(* CoDeSys 2.3 project: cy-wg-05-005.pro *)
(* Title: cy-wg-05 - ClevergyAS *)
(* Author: Andrea Ravasio *)
(* Libraries: Standard.lib 2.12.10 14:48:34, Util.lib 18.5.10 15:14:28, Visual.lib 2.12.10 14:48:34, WagoLibIdent.lib 25.2.13 11:12:16, WagoLibStatus.lib 2.12.10 14:48:32, SysLibFile.lib 2.12.10 14:48:34, SysLibRtc.lib 2.12.10 14:48:32, SysLibSockets.lib 10.2.11 09:20:54, SysLibEvent.lib 2.12.10 14:48:34, SysLibPlcCtrl.lib 2.12.10 14:48:32, SysLibCallback.lib 2.12.10 14:48:32, mod_com.lib 2.12.10 14:48:32, SerComm.lib 31.5.11 08:54:36, Serial_Interface_01.lib 22.4.13 12:50:14, Modb_l05.lib 22.4.13 12:50:12, MBus_03.lib 9.2.13 17:51:58 *)

(* PLC configuration (modules and I/O channels)
K-Bus [K_Bus] node 0, in %IB0 out %QB0
  0750-0402 4 DI 24 V DC 3.0ms [Type_1_4_Channels] node 0, in %IB8 out %QB8 {INTTypePAAssignment = PLC; INTTypeModule = plugged}
    VPN_OUT2 AT %IX4.0 [BOOLOnX_I] Ch_1 Digital input
    KEY_QE_ST AT %IX4.1 [BOOLOnX_I] Ch_2 Digital input
    AT %IX4.2 [BOOLOnX_I] Ch_3 Digital input
    AT %IX4.3 [BOOLOnX_I] Ch_4 Digital input
  0750-0504 4 DO 24V DC 0.5A [Type_10_4_Channels] node 1, in %IB8 out %QB8 {INTTypePAAssignment = PLC; INTTypeModule = plugged}
    AT %QX4.0 [BOOLOnX_Q] Ch_1 Digital output
    AT %QX4.1 [BOOLOnX_Q] Ch_2 Digital output
    TEST1 AT %QX4.2 [BOOLOnX_Q] Ch_3 Digital output
    TEST2 AT %QX4.3 [BOOLOnX_Q] Ch_4 Digital output
  0750-0653/0003-0000#03 RS485 Interface (Adjustable), 3 Bytes [Type_21_1_Channels] node 2, in %IB4 out %QB4 {INTTypePAAssignment = PLC; INTTypeModule = plugged}
    AT %IX0.0 [BOOLOnX_I] Transmission acknowledgement
    AT %IX0.1 [BOOLOnX_I] Reception request
    AT %IX0.2 [BOOLOnX_I] Initialization acknowledgement
    AT %IX0.3 [BOOLOnX_I] Input buffer is full
    AT %IX0.4 [BOOLOnX_I] Number of received characters Bit 0
    AT %IX0.5 [BOOLOnX_I] Number of received characters Bit 1
    AT %IX0.6 [BOOLOnX_I] Number of received characters Bit 2
    AT %IB1 [BYTEOnB_I] Input data Byte 0
    AT %IB2 [BYTEOnB_I] Input data Byte 1
    AT %IB3 [BYTEOnB_I] Input data Byte 2
    AT %QX0.0 [BOOLOnX_Q] Transmission request
    AT %QX0.1 [BOOLOnX_Q] Reception acknowledgement
    AT %QX0.2 [BOOLOnX_Q] Initialization request
    AT %QX0.4 [BOOLOnX_Q] Number of characters Bit 0
    AT %QX0.5 [BOOLOnX_Q] Number of characters Bit 1
    AT %QX0.6 [BOOLOnX_Q] Number of characters Bit 2
    AT %QB1 [BYTEOnB_Q] Output data Byte 0
    AT %QB2 [BYTEOnB_Q] Output data Byte 1
    AT %QB3 [BYTEOnB_Q] Output data Byte 2
  0750-0650/0003-0000#03 RS 232 C Interface (Adjustable), 3 Byte [Type_21_1_Channels] node 0, in %IB4 out %QB4 {INTTypePAAssignment = PLC; INTTypeModule = plugged}
    AT %IX2.0 [BOOLOnX_I] Transmission acknowledgement
    AT %IX2.1 [BOOLOnX_I] Reception request
    AT %IX2.2 [BOOLOnX_I] Initialization acknowledgement
    AT %IX2.3 [BOOLOnX_I] Input buffer is full
    AT %IX2.4 [BOOLOnX_I] Number of received characters Bit 0
    AT %IX2.5 [BOOLOnX_I] Number of received characters Bit 1
    AT %IX2.6 [BOOLOnX_I] Number of received characters Bit 2
    AT %IB5 [BYTEOnB_I] Input data Byte 0
    AT %IB6 [BYTEOnB_I] Input data Byte 1
    AT %IB7 [BYTEOnB_I] Input data Byte 2
    AT %QX2.0 [BOOLOnX_Q] Transmission request
    AT %QX2.1 [BOOLOnX_Q] Reception acknowledgement
    AT %QX2.2 [BOOLOnX_Q] Initialization request
    AT %QX2.4 [BOOLOnX_Q] Number of characters Bit 0
    AT %QX2.5 [BOOLOnX_Q] Number of characters Bit 1
    AT %QX2.6 [BOOLOnX_Q] Number of characters Bit 2
    AT %QB5 [BYTEOnB_Q] Output data Byte 0
    AT %QB6 [BYTEOnB_Q] Output data Byte 1
    AT %QB7 [BYTEOnB_Q] Output data Byte 2
Fieldbus variables [FB_VARS] node 1, in %IB0 out %QB0
Flag variables [FLAG_VARS] node 2, in %IB0 out %QB0
Modbus-Master [MB_MASTER] node 3, in %IB0 out %QB0
*)

(* Global variable list: Global_Constants *)
VAR_GLOBAL CONSTANT

	Plant_NAME			: STRING :='cySN:5 cyVER:5 - Gavazzeni C Energetiche';
	Plant_SN			: DWORD  :=5;  		(* S/N Impianto di telecontrollo *)
	Plant_SW_VER		: WORD   :=5;		(* Versione SW installata *)

	(* Parameters *)
	Plant_DefaultTAmb	: INT	:=100;		(* [.1°C] Temperatura ambiente di default in caso di rottura sonda *)
	Plant_MaxRunTAmb	: INT   :=250; 		(* [.1°C] Temperatura ambiente massima funzionamento impianto *)
	Plant_AntiFreezeTAmb: INT   :=-40;		(* [.1°C] Antifreeze temperature, start circulators *)
	Plant_VRD_TAlarm	: INT   :=450; 		(* [.1°C] Temperatura di allarme VRD, blocco *)
	Plant_VRD_TMax		: INT   :=430; 		(* [.1°C] Setpoint massimo per uscita VRD *)
	Plant_VRD_TDefault	: INT	:=300;		(* [.1°C] Temperatura di default in caso di errore climatica *)
	Plant_CirOffDelay	: TIME	:=T#15m;	(* (Def.T#15m) Ritardo spegnimento pompe per ricircolo caldaia *)
	Plant_MaxWaterLoss	: WORD  :=2;		(* [lt/h] Massima perdita del circuito *)

	(* Filesystem *)
	FilesPath  			: STRING :='S:\';

	(* TCP Logger *)
	Logger_SERVER		: STRING:='';
	Logger_IP			: STRING:='192.168.100.3';
	Logger_PORT			: WORD  :=80;
	Logger_GETSTART		: STRING:='GET /cygmsrv/hsgm.ashx?';
	Logger_GETEND		: STRING:='$R$N$R$N';
	Logger_CHECK		: STRING:='True';
	Logger_CRLF			: STRING:='$R$N';
	Logger_DataFile		: STRING:='S:\LOG.DAT';
	Logger_DataFileOld	: STRING:='S:\LOG.BCK';
	Logger_IndexFile	: STRING:='S:\LOG.IDX';
	Logger_ConnRetries	: BYTE:=5;
	Logger_RecoverMsgs	: BYTE:=25;

	(* TCP Remote *)
	Remote_PORT			: WORD  :=10;
	Remote_WELCOME		: STRING:='Connected$R$N';
	Remote_OK			: STRING:='OK$R$N';
	Remote_ERROR		: STRING:='ERROR$R$N';

	(* TCP Sockets *)
	MAX_SEND_TCP_SERVER					 : DWORD:=1500;(*60000*)
	MAX_RECEIVE_TCP_SERVER				 : DWORD:=3000;
	MAX_RECEIVE_TCP_SERVER_SOCKET	 	 : DWORD:=1500;
	MAX_SEND_TCP_CLIENT					 : DWORD:=1500;(*15000*)
	MAX_RECEIVE_TCP_CLIENT				 : DWORD:=1500;
	MAX_RECEIVE_TCP_CLIENT_SOCKET		 : DWORD:=1500;
	MAX_RECEIVE_UDP_SERVER				 : INT  :=1472;
	MAX_RECEIVE_UDP_CLIENT				 : INT  :=1472;
	CONNECT_WATCHDOG_TIME				 : TIME :=t#10s;

END_VAR

(* Global variable list: Global_Retain *)
VAR_GLOBAL RETAIN PERSISTENT
	Mode_Manual : BOOL := FALSE;
END_VAR

(* Global variable list: Global_Variables *)
VAR_GLOBAL

	SYS    : typ_SYS;

	MODB01 : obj_MODBUS						:= ( ID:=1 , COM:=2, BAUDRATE:=BAUD_9600, RS485:=TRUE );
	GAS01  : obj_MODBUS_ELGAS_MINIELCOR		:= ( ID:=1 , ADDRESS:=1 );

	MBUS01 : obj_MBUS						:= ( ID:=1 , COM:=3, BAUDRATE:=BAUD_2400 );
	CTB01  : obj_MBUS_CTB_SHARKY775			:= ( ID:=1 , ADDRESS:=16#51311891 );
	CTB02  : obj_MBUS_CTB_SHARKY775			:= ( ID:=2 , ADDRESS:=16#51311893 );
	CTB03  : obj_MBUS_CTB_SHARKY775			:= ( ID:=3 , ADDRESS:=16#51311892 );
	CTB04  : obj_MBUS_CTB_SHARKY775			:= ( ID:=4 , ADDRESS:=16#51038660 );

	Logger : typ_Logger;

	(**** SIMULATION ONLY ****)
(*	VPN_ST2		:BOOL:=TRUE;
	KEY_QE_ST	:BOOL:=TRUE;
*)

END_VAR

(* Data type in Logger *)
TYPE en_Logger_ErrLev :
(
	EL_Log			:=0,
	EL_Wrn			:=1,
	EL_Alarm		:=2,
	EL_AlarmStop	:=3
);
END_TYPE

(* Data type in Logger *)
TYPE en_Logger_Status :
(
	S_Logger_UNKNOWN := 0,
	S_Logger_IDLE,
	S_Logger_WAITCONN,
	S_Logger_WAITTX,
	S_Logger_WAITRESP,
	S_Logger_ERROR
);
END_TYPE

(* Data type *)
TYPE en_SYS_Objects :
(
	EO_SYS		:=0,  (* PLC *)
	EO_VPN		:=1,  (* VPN *)
	EO_DOOR		:=2,  (* Door & access control *)

	EO_CAL		:=10, (* Caldaia *)
	EO_CIR		:=11, (* Circolatore *)
	EO_CRON		:=12, (* Crono-termostato *)
	EO_VRD		:=13, (* Valvola miscelatore pannelli *)
	EO_CTL		:=14, (* Contalitri *)
	EO_CTB		:=15, (* Contabilizzatore *)
	EO_TPV		:=16, (* Temperature probes values *)
	EO_PPV		:=17, (* Pressure probes values *)
	EO_PBV		:=18, (* Over-Pressure Alarms *)
	EO_TBV		:=19, (* Over-Temperature Alarms *)
	EO_PMV		:=20, (* Under-Pressure Alarms *)
	EO_GRU		:=21, (* Gruppo termico *)
	EO_PDC		:=22, (* Pompa di calore *)
	EO_SOL		:=23, (* Pannello solare termico *)
	EO_ESOL		:=24, (* Pannello solare fotovoltaico *)
	EO_GAS		:=25, (* Contatore GAS *)
	EO_PORT		:=26, (* Misuratore di portata *)
	EO_FPV		:=27, (* Flow probes value *)
	EO_ANZ		:=28, (* Analizzatore di rete elettrica *)

	EO_LON		:=1000, (* Bus - LON *)
	EO_MODBUS	:=1001, (* Bus - MODBUS *)
	EO_MBUS		:=1002  (* Bus - M-BUS *)
);
END_TYPE

(* Data type *)
TYPE en_SYS_Status :
(
	S_UNKNOWN  := 0,
	S_STARTUP,
	S_INIT_RTC,
	S_INIT_VAR,
	S_AUTOTEST,
	S_RUNNING,
	S_SHUTDOWN,
	S_HALT
);
END_TYPE

(* Data type in Plant_Objects *)
TYPE typ_Clima : (* CURVA CLIMATICA *)
STRUCT
	InitOK:		BOOL;
	Points: 	ARRAY [0..10] OF POINT;
END_STRUCT
END_TYPE

(* Data type in Plant_Objects *)
TYPE typ_Cron_Calendar :
STRUCT
	Profile		: ARRAY[0..384] OF BYTE;
END_STRUCT
END_TYPE

(* Data type in Plant_Objects *)
TYPE typ_Cron_Jolly :
STRUCT
	Start		: DT;
	End			: DT;
	Temp		: WORD;
	Flags		: WORD; (* B0:Enabled B1..B15:Unused *)
END_STRUCT
END_TYPE

(* Data type in Plant_Objects *)
TYPE typ_Cron_Profile :
STRUCT
	Flags		: WORD;
	Setpoint	: ARRAY [0..95] OF WORD;
END_STRUCT
END_TYPE

(* Data type in Logger *)
TYPE typ_Logger :
STRUCT
	Status		: en_Logger_Status;

	SendReq		: BOOL;
	SendIdx		: DWORD;
	SendData	: ARRAY [0..MAX_SEND_TCP_CLIENT] OF BYTE;
	SendLen		: DINT;

	TData		: ARRAY [0..MAX_SEND_TCP_CLIENT] OF BYTE;
	TLen		: DINT;

	LastIdxPos	: DWORD;

	(* Temporary variables used by objects *)
	s1			: STRING(256);
	i1			: WORD;

END_STRUCT
END_TYPE

(* Data type in Plant_Objects *)
TYPE typ_MODBUS_ABB_DMTME72 :
STRUCT
	V_3P		: DWORD; (* V *)
	V_L1N		: DWORD;
	V_L2N		: DWORD;
	V_L3N		: DWORD;
	V_L1L2		: DWORD;
	V_L2L3		: DWORD;
	V_L3L1		: DWORD;
	I_3P		: DWORD; (* 10^-3 A *)
	I_L1		: DWORD;
	I_L2		: DWORD;
	I_L3		: DWORD;
	PF_3P		: DINT;	 (* 10^-3 *)
	PF_L1		: DINT;
	PF_L2		: DINT;
	PF_L3		: DINT;
	COS_3P		: DINT;
	COS_L1		: DINT;
	COS_L2		: DINT;
	COS_L3		: DINT;
	VA_3P		: DWORD; (* VA *)
	VA_L1		: DWORD;
	VA_L2		: DWORD;
	VA_L3		: DWORD;
	P_3P		: DWORD; (* W *)
	P_L1		: DWORD;
	P_L2		: DWORD;
	P_L3		: DWORD;
	Q_3P		: DWORD; (* VAr *)
	Q_L1		: DWORD;
	Q_L2		: DWORD;
	Q_L3		: DWORD;

	WH_3P		: DWORD; (* 10^-2 Wh *)
	VARH_3P		: DWORD; (* 10^-2 VArh *)
	FREQ		: DWORD; (* 10^-3 Hz *)

	I_L1_Max	: DWORD;
	I_L2_Max	: DWORD;
	I_L3_Max	: DWORD;
	P_3P_Max	: DWORD;
	Q_3P_Max	: DWORD;
	P_3P_Avg15m	: DWORD;

END_STRUCT
END_TYPE

(* Data type in Plant_Objects *)
TYPE typ_MODBUS_ELGAS_MINIELCOR :
STRUCT
	Vb			: ARRAY [0..3] OF WORD;	(* m^3 *)
	Vm			: DWORD;				(* m^3 *)
	P			: REAL;					(* bar *)
	T			: REAL;					(* °C *)
	C			: REAL;
	Vbs			: ARRAY [0..3] OF WORD;	(* m^3 *)
	Vb_d_d		: ARRAY [0..3] OF WORD;	(* m^3 *)
	Vb_d_m		: ARRAY [0..3] OF WORD;	(* m^3 *)
	Vm_d_d		: DWORD;				(* m^3 *)
	Q			: REAL;					(* m^3/h *)
	Qb			: REAL;					(* m^3/h *)

	BC_EVC		: REAL;			(* % *)
	BV_EVC		: REAL;			(* V *)
	D_Err		: WORD;			(* 0:OK, 1:FAIL *)
	Status		: DWORD;		(* Status bits *)

END_STRUCT
END_TYPE

(* Data type in Plant_Objects *)
TYPE typ_MODBUS_FRER_IQ96U2 :
STRUCT
	V_L1N		: DWORD; (* 10^-3 V *)
	V_L2N		: DWORD;
	V_L3N		: DWORD;
	V_L1L2		: DWORD;
	V_L2L3		: DWORD;
	V_L3L1		: DWORD;
	I_L1		: DWORD; (* 10^-3 I *)
	I_L2		: DWORD;
	I_L3		: DWORD;
	FREQ		: DWORD; (* 10^-3 Hz *)
	P_3P		: DWORD; (* W *)
	Q_3P		: DWORD; (* VAr *)
	PF_3P		: DINT;	 (* 10^-3 *)
	WH_3P		: DWORD; (* Wh *)
	VARH_3P		: DWORD; (* VArh *)
	MULT		: DWORD;

	WH_3P_NEG	: DWORD; (* Wh *)
	VARH_3P_NEG : DWORD; (* VArh *)
	S_3P		: DWORD; (* VA *)

	PF_L1		: DWORD; (* 10^-3 *)
	PF_L2		: DWORD; (* 10^-3 *)
	PF_L3		: DWORD; (* 10^-3 *)

	P_3P_Max	: DWORD;
	P_3P_Avg15m	: DWORD;
	I_L1_Max	: DWORD;
	I_L2_Max	: DWORD;
	I_L3_Max	: DWORD;
	I_L1_Avg15m	: DWORD;
	I_L2_Avg15m	: DWORD;
	I_L3_Avg15m	: DWORD;

END_STRUCT
END_TYPE

(* Data type in Plant_Objects *)
TYPE typ_MODBUS_VAR : (* Gestione parametri MODBUS *)
STRUCT
	SlaveAddress	: BYTE;
	FunCode			: BYTE;
	FunAddress		: WORD;
	Refresh_Time	: BYTE; (* 0:No refresh x:Refresh in seconds *)
	Refresh_Cnt		: BYTE; (* INTERNAL *)
	Variable		: POINTER TO WORD;
	Variable_Size	: BYTE;
	Variable_Mirror : WORD; (* INTERNAL [Force refresh on read variables when <>0] *)
END_STRUCT
END_TYPE

(* Data type *)
TYPE typ_SYS :
STRUCT
	Status			: en_SYS_Status;
	Warning			: BOOL;
	Alarm			: BOOL;
	AlarmStop		: BOOL;

	Time_LogString	: STRING;
	Time_Year		: WORD;
	Time_Month		: BYTE;
	Time_Day		: BYTE;

	Time_CT_DT		: DT;
	Time_CT_Day		: WORD;
	Time_CT_Quarter	: BYTE;

	LastLogs_Idx	: BYTE;
	LastLogs_Dat	: ARRAY[0..5] OF STRING;
	LastLogs_Msg	: ARRAY[0..5] OF STRING;

END_STRUCT
END_TYPE

(* POU PLC_PRG, ST *)
PROGRAM PLC_PRG
VAR
	Timer1: TON; (* Fast controls tick *)
	Timer2: TON; (* Plant control tick *)
	Timer3: TON; (* Logger timer *)
END_VAR
(******************************************************************************
 ****                           MAIN TASK CODE                             ****
 ******************************************************************************

	Network setup:
		IP  = 192.168.100.2 | MSK = 255.255.255.0
		GW	= 192.168.100.1 | DNS = 192.168.100.1
		SNTP = 193.204.114.232 (3600s) ==> 192.168.100.3

*)

(*==============================*)
(*===== Main status machine ====*)
(*==============================*)
Main_Stm();

(*==============================*)
(*== Running cycle operations ==*)
(*==============================*)
IF SYS.Status>S_INIT_VAR THEN

	(* Execute MODBUS01 process *)
	MODB01();
	GAS01( MODBUS:=MODB01 );

	(* Execute MBUS01 process *)
	MBUS01();
	CTB01( MBUS:=MBUS01 );
	CTB02( MBUS:=MBUS01 );
	CTB03( MBUS:=MBUS01 );
	CTB04( MBUS:=MBUS01 );

END_IF

(*==============================*)
(*== System cycle operations ===*)
(*==============================*)
(* Execute TCP processes *)
Logger_Proc();
Remote_Proc();
(* Update user led *)
USRLED_Update();
(* Execute Cron Editor commands *)
(*CronEd(); *)
(* External resources *)
(*	IF NOT TPV01.ERR THEN T_AMB:=T_S01;
ELSIF NOT TPV05.ERR THEN T_AMB:=GRU01.TAmb;
ELSE 					 T_AMB:=Plant_DefaultTAmb;
END_IF *)

(**** SIMULATION ONLY ****)
(*...*)
END_PROGRAM
ACTION Main_Stm:
CASE Sys.Status OF

	S_STARTUP:
		Sys.Status:=S_INIT_RTC;

	S_INIT_RTC:
		(* Check RTC and update from network *)
		RTC_Update();
		(* Check time *)
		IF Sys.Time_Year>2000 THEN
			Sys.Status:=S_INIT_VAR;
		END_IF

	S_INIT_VAR:
		LogEv(EL_Wrn,EO_SYS,0,1,CONCAT('System_startup_v',WORD_TO_STRING(Plant_SW_VER)));
		Sys.Status:=S_RUNNING;

	S_RUNNING:
		Timer1(IN:=NOT Timer1.Q,PT:=T#50ms);
		IF Timer1.Q THEN
			(* Update meters *)

			(* Update system checks *)
			SYS_Proc();
		END_IF

		Timer2(IN:=NOT Timer2.Q,PT:=T#500ms);
		IF Timer2.Q THEN
			(* Read current date/time *)
			RTC_Update();
			(* Execute plant operations *)

			(* Test toggle *)
			IF TEST1 THEN TEST1:=FALSE; ELSE TEST1:=TRUE; END_IF
		END_IF

		Timer3(IN:=NOT Timer3.Q,PT:=T#5m);
		IF Timer3.Q THEN
			(* Trig logger *)
			LogTrig();
			(* Execute temporary CSV logger *)
			(*CSV_Log();*)
		END_IF

	S_SHUTDOWN:
		(* Stop sistema *)
		Sys.Status:=S_STARTUP;

	S_HALT:
		(* Aspetta uscita manuale *)
		Sys.Status:=S_STARTUP;

ELSE
	Sys.Status:=S_STARTUP;
END_CASE;
END_ACTION

(* POU TCP_Logger/Logger_Proc, ST *)
PROGRAM Logger_Proc
VAR
	c1:         	TCPCLIENT;

	Open:	    	BOOL;
	IpAddr:			DWORD;
	InetAddr:		DWORD;
	Connected:  	BOOL;
	Error:      	DINT;
	TxTrig:     	BOOL;
	RxData:			ARRAY [0..MAX_RECEIVE_TCP_CLIENT] OF BYTE;
	RxLen:			DINT;

	Retry:			BYTE;	(* Counter for connection retries *)
	Recovered:		BYTE;	(* Counter for recovered unsent messages *)

	i:				DINT;
	pos:			DWORD;
	hFile:			DWORD;

END_VAR
(*=== State machine ===*)
CASE Logger.Status OF

	S_Logger_UNKNOWN:
		(* Startup *)
		Logger.SendReq:=FALSE;
		Open:=FALSE;
		Logger.Status:=S_Logger_IDLE;

	S_Logger_IDLE:
		(* Wait request *)
		IF Logger.SendReq THEN
			(* Resolve server name or use static IP *)
			IF LEN(Logger_SERVER)=0 THEN
				InetAddr:=SysSockInetAddr(Logger_IP);
			ELSE
				IpAddr:=SysSockGetHostByName(ADR(Logger_SERVER));
				DWORDSWAP(pIn:=ADR(IpAddr), pOut:=ADR(InetAddr));
			END_IF
			TxTrig:=FALSE;
			RxLen:=0;
			(* Open connection *)
			Open:=TRUE;
			Logger.Status:=S_Logger_WAITCONN;
		END_IF

	S_Logger_WAITCONN:
		(* Wait connection *)
		IF Connected THEN
			(* Send data *)
			TxTrig:=TRUE;
			Logger.Status:=S_Logger_WAITTX;
		END_IF
		IF Error>0 THEN
			Open:=FALSE;
			Logger.Status:=S_Logger_ERROR;
		END_IF

	S_Logger_WAITTX:
		(* Wait transmission *)
		IF NOT TxTrig THEN
			Logger.Status:=S_Logger_WAITRESP;
		END_IF
		IF Error>0 THEN
			Open:=FALSE;
			Logger.Status:=S_Logger_ERROR;
		END_IF

	S_Logger_WAITRESP:
		(* Wait response *)
		IF Connected=FALSE (* OR TIMEOUT!! *) THEN
			Open:=FALSE;
			(* Check response *)
			IF RxLen>=4 AND CHKSTRING(pString:=ADR(RxData), pPattern:=ADR(Logger_CHECK)) THEN
				Logger.SendReq:=FALSE;
				Retry:=0;
				(* Check unsent messages to flush *)
				IF Recovered<Logger_RecoverMsgs THEN
					MsgChk();
					IF Logger.SendReq=TRUE THEN
						Recovered:=Recovered+1;
					ELSE
						Recovered:=0;
					END_IF
				ELSE
					Recovered:=0;
				END_IF
				Logger.Status:=S_Logger_IDLE;
			ELSE
				Logger.Status:=S_Logger_ERROR;
			END_IF
		END_IF

	S_Logger_ERROR:
		(* Connection error or send failure *)
		Retry:=Retry+1;
		IF Retry>Logger_ConnRetries THEN
			(* Save message as unsent *)
			MsgSave();
			Logger.SendReq:=FALSE;
			Retry:=0;
		END_IF
		Logger.Status:=S_Logger_IDLE;

ELSE
	Logger.Status:=S_Logger_UNKNOWN;
END_CASE


(*=== Execute client lib ===*)
c1(
	xOpenConnection			:= Open,
	dwInetAddr 				:= InetAddr,
	wPortNumber				:= Logger_PORT,
	ptSendData				:= ADR(Logger.SendData),
	diSendCount				:= Logger.SendLen,
	tConnectWatchdogTime	:= t#10s,
	xStartSend				:= TxTrig,
	aReceiveBuffer			:= RxData,
	diReceiveCount			:= RxLen,
	xConnected				=> Connected,
	diError					=> Error
);

(*=== Process Rx data ===*)
(*IF RxLen>0 THEN
	RxLen:=0;
END_IF*)
END_PROGRAM
ACTION MsgChk:
(* Open index file *)
hFile:=SysFileOpen(Logger_IndexFile,'r');
IF hFile=0 THEN
	RETURN;
END_IF
(* Search oldest message to recover *)
SysFileSetPos(hFile,Logger.LastIdxPos);
Logger.SendLen:=0;
REPEAT
	SysFileRead(hFile, ADR(Logger.SendIdx), SIZEOF(Logger.SendIdx));
	pos:=SysFileGetPos(hFile);
	SysFileRead(hFile, ADR(Logger.SendLen), SIZEOF(Logger.SendLen));
UNTIL
	SysFileEOF(hFile) OR Logger.SendLen<>0
END_REPEAT
SysFileClose(hFile);
(* Delete index file when all messages are recovered *)
IF Logger.SendLen=0 THEN
	Logger.LastIdxPos:=0;
	SysFileDelete(Logger_IndexFile);
	RETURN;
END_IF
(* Recover message data *)
hFile:=SysFileOpen(Logger_DataFile,'r');
IF hFile<>0 THEN
	SysFileSetPos(hFile,Logger.SendIdx);
	SysFileRead(hFile,ADR(Logger.SendData),Logger.SendLen);
	Logger.SendReq:=TRUE;
	SysFileClose(hFile);
END_IF
(* Clear index entry *)
hFile:=SysFileOpen(Logger_IndexFile,'a');
IF hFile<>0 THEN
	SysFileSetPos(hFile,pos);
	i:=0;
	SysFileWrite(hFile, ADR(i), 4);
	Logger.LastIdxPos:=SysFileGetPos(hFile);
	SysFileClose(hFile);
END_IF
END_ACTION
ACTION MsgSave:
(* Add log position in recovery indexes *)
hFile:=SysFileOpen(Logger_IndexFile,'a');
SysFileWrite(hFile, ADR(Logger.SendIdx), SIZEOF(Logger.SendIdx));
SysFileWrite(hFile, ADR(Logger.SendLen), SIZEOF(Logger.SendLen));
SysFileClose(hFile);
END_ACTION

(* POU Utils Functions/TCPCLIENT, ST *)
FUNCTION_BLOCK TCPCLIENT
(***********************************************************************************************************	*)
(* Version: 1.3b                        			          													*)
(* Date: 28.10.2014                   				          							            			*)
(***********************************************************************************************************	*)
(* WAGO Kontakttechnik GmbH Hansastr. 27 32423 Minden(Westf.)													*)
(* Tel. +0049 571/887-0 Fax. +0049 571/887-0																	*)
(* Author: VB																									*)
(***********************************************************************************************************	*)
(*Description:	A TCP client to read and write data with additional connection watchdog							*)
(*History:																										*)
(*Version 1.3b: 28.10.2014: Use DWORD address for IP (Andrea Ravasio)											*)
(*Version 1.3: 11.02.2011: Changes according to 750-880/881											 			*)
(*Version 1.2: 29.08.2007 Bugfix TCP Client																		*)
(*Version 1.1: 15.01.2007 Changes according to FW11																*)
(*Version 1.0: 09.03.2006 Release																				*)
(***********************************************************************************************************	*)
VAR CONSTANT
	STATE_CREATE     				 : BYTE:= 0;
	STATE_OPEN     					 : BYTE:= 1;
	STATE_IOCTL    					 : BYTE:= 2;
	STATE_CONNECT     				 : BYTE:= 10;
	STATE_TX       					 : BYTE:= 20;
	STATE_RX       					 : BYTE:= 30;
	STATE_CLOSE    					 : BYTE:= 40;
	STATE_ERROR_TRAP			     : BYTE:= 200;
END_VAR

VAR_INPUT
	xOpenConnection					: BOOL;
	dwInetAddr						: DWORD; (* <== Use SysSockInetAddr() value or
													swapped bytes order of SysSockGetHostByName() value *)
	wPortNumber						: WORD;
	ptSendData						: POINTER TO ARRAY[0..MAX_SEND_TCP_CLIENT] OF BYTE;
	diSendCount						: DINT;
	tConnectWatchdogTime		    : TIME := t#10s;
END_VAR
VAR_OUTPUT
	xConnected						: BOOL;
	diError 						: DINT := 0;
END_VAR
(* ErrorCodes -----------------------------------------
	16#8001 => No socket descriptor available 
	16#8002 => SysSockSend returns -1 
	16#8003 => Socket was "gracefully closed" 
	16#8004 => switching to none blocking mode fails
	16#8005 => SysSockClose() returns FALSE 
    16#8006 => SysSockConnect() fails
    16#8007 => SysSockSend() fails
	16#8008 => error state machine 
	16#8009 => timeout while waiting for data from server 
------------------------------------------------------------*)
VAR_IN_OUT
	xStartSend							: BOOL;
	aReceiveBuffer						: ARRAY [0..MAX_RECEIVE_TCP_CLIENT] OF BYTE;
	diReceiveCount						: DINT;
END_VAR
VAR
	m_State								: BYTE := 0;
	m_ReceiveBuffer						: ARRAY [0..MAX_RECEIVE_TCP_CLIENT_SOCKET] OF BYTE;
	m_Socket							: DINT;
	m_AddressInfo						: SOCKADDRESS;
	m_BytesReceived						: DINT;
	m_diReturn							: DINT;
	m_xReturn							: BOOL;
	m_IoCtlParameter  					: DINT := 1; (* IOCTL-Parameter for non-blocking mode of sockets *)
	i									: INT;
	T_Connect							: TON;
	m_count								: DINT;
	diOption							: DINT := 1;
	m_Blocking   						: DINT := 0;
END_VAR
IF xOpenConnection THEN
	(* State maschine *)
	CASE  m_State OF

	(* -------------------------------------------------------------------------*)
	STATE_CREATE:
			(* create socket descriptor*)
			m_Socket := SysSockCreate(diAddressFamily	:= SOCKET_AF_INET,
													 diType		:= SOCKET_STREAM,
													 diProtocol := SOCKET_IPPROTO_TCP);
			IF m_Socket >= 0 THEN
			(*Set Push-Bit*)
				IF ADR(%MW0)=16#30000000  OR ADR(%MW0)=16#20000000 THEN (*841 or 881*)
					SysSockSetOption(
						diSocket:=m_Socket,
						diLevel:=6,
						diOption:=SOCKET_TCP_NODELAY,
						pOptionValue:=ADR(diOption),
						diOptionLength:=SIZEOF(diOption));
				ELSE
						;
				END_IF
				m_State := STATE_IOCTL; (* succesful *)
			ELSE
				diError := 16#8001;  (* no socket descriptor available *)
				m_State := STATE_ERROR_TRAP;
			END_IF

	(* -------------------------------------------------------------------------*)
	STATE_IOCTL: (* change  socket mode  to none blocking *)
		m_diReturn := SysSockIoctl( m_Socket, SOCKET_FIONBIO, ADR(m_IoCtlParameter));
		IF m_diReturn <> 0 THEN
			m_AddressInfo.sin_family := SOCKET_AF_INET;
			m_AddressInfo.sin_port := SysSockNtohs(wPortNumber);
			m_AddressInfo.sin_addr := dwInetAddr;
			m_State := STATE_CONNECT;
		ELSE
			diError := 16#8004;  (* switching to none blocking mode fails *)
			m_State := STATE_ERROR_TRAP;
		END_IF


	(* -------------------------------------------------------------------------*)
	STATE_CONNECT: (* connect with server *)
		T_Connect(IN:=TRUE , PT:=tConnectWatchdogTime);(*activate watchdog for establishing connection to a server*)
		m_xReturn := SysSockConnect ( m_Socket, ADR(m_AddressInfo),  SIZEOF(m_AddressInfo));
		IF m_xReturn THEN (* succesful *)
			IF xStartSend THEN
				m_State := STATE_TX;(*transmit data*)
			ELSE
				m_State := STATE_RX;(*wait for data from server*)
			END_IF
			xConnected:=TRUE;
			T_Connect(IN:=FALSE);
		ELSE
			IF T_Connect.Q THEN
				diError := 16#8006;  (* connect fails *)
				xConnected:=FALSE;
				T_Connect(IN:=FALSE);
				m_State := STATE_ERROR_TRAP;
				SysSockClose( m_Socket);
			ELSE
				m_State := STATE_CONNECT;(*client still  tries to set up connection*)
			END_IF
		END_IF


	STATE_TX:	 (* send TCP-message *)
		m_diReturn := SysSockSend(diSocket := m_Socket,
								  pbyBuffer := ADR(ptSendData^[0]),
								  diBufferSize := diSendCount-m_count,
								  diFlags := 0);

		CASE m_diReturn OF
		-1:	(* ERROR *)
			T_Connect(IN:=TRUE , PT:=CONNECT_WATCHDOG_TIME);(*activate watchdog to check communication*)
			IF t_Connect.Q THEN
				diError := 16#8007;
				T_Connect(IN:=FALSE);
				m_State:=STATE_CLOSE;
			END_IF
		0: (* socket was "gracefully closed" *)
			m_State := STATE_CLOSE;
			diError := 16#8003;
		ELSE (* succesful *)
			m_count:=m_count+m_diReturn;
			IF m_count>=diSendCount THEN
				diError := 16#0000;
				m_State := STATE_RX;
				m_count:=0;
				xStartSend:=FALSE;
			END_IF
			T_Connect(IN:=FALSE);
		END_CASE

	(* -------------------------------------------------------------------------*)
	STATE_RX: (* process receive data *)
			m_BytesReceived := SysSockRecv(	diSocket 	:= m_Socket,
										pbyBuffer 	:= ADR(m_ReceiveBuffer),		(* Address of receive buffer *)
										diBufferSize:= SIZEOF(m_ReceiveBuffer),
										diFlags		:= 0);

			CASE m_BytesReceived OF
			-1:	(* No data available or error occured *)
				T_Connect(IN:=TRUE , PT:=tConnectWatchdogTime);(*activate watchdog to check communication*)
				IF t_Connect.Q THEN
					diError:=16#8009;
					T_Connect(IN:=FALSE);
					m_State:=STATE_CLOSE;
				END_IF
				IF xStartSend THEN
					m_State:=STATE_TX	;(* WAIT IN THIS STATE  and check for arriving data or new send command*)
				END_IF;
			0: (* socket was "gracefully closed"  *)
				m_State:=STATE_CLOSE;
				diError := 16#8003;
			ELSE (* succesful *)
				diError := 16#0000;
				T_Connect(IN:=FALSE);
				(* Copy received data into receive buffer *)
				FOR i:= 0 TO DINT_TO_INT(m_BytesReceived	)-1 DO
					aReceiveBuffer[diReceiveCount]:= m_ReceiveBuffer[i];
					diReceiveCount:=(diReceiveCount+1) MOD SIZEOF(aReceiveBuffer);
				END_FOR

			END_CASE

	(* -------------------------------------------------------------------------*)
	STATE_CLOSE : (* close socket *)
		IF ADR(%MW0)=16#30000000  OR ADR(%MW0)=16#20000000 THEN (*841 or 881*)
			;
		ELSE
			SysSockShutdown(m_Socket, 0);;(*870*)
		END_IF
		m_xReturn := SysSockClose( m_Socket);
		m_Socket := -1;
		m_State := 0; (* succesful *)
		xConnected:=FALSE;
		T_Connect(IN:=FALSE);
	(* -------------------------------------------------------------------------*)
	STATE_ERROR_TRAP: (* error handling *)
		xConnected:=FALSE;

	ELSE  (* Bad FSM code trap  *)
			m_State:= STATE_ERROR_TRAP;
			diError:= 16#8008;
	END_CASE

ELSE(*close connection*)
	IF m_Socket >= 0 THEN
		IF ADR(%MW0)=16#30000000  OR ADR(%MW0)=16#20000000 THEN (*841 or 881*)
			;
		ELSE
			SysSockShutdown(m_Socket, 0);;(*870*)
		END_IF
		SysSockClose( m_Socket);
	END_IF
	m_Socket := -1;
	diError := 16#0000;
	m_State := STATE_CREATE;
	xConnected:=FALSE;
	T_Connect(IN:=FALSE);
END_IF
END_FUNCTION_BLOCK

(* POU Utils Functions/DWORDSWAP, ST *)
FUNCTION DWORDSWAP:BOOL
VAR_INPUT
	pIn:POINTER TO ARRAY[1..4] OF BYTE;
	pOut:POINTER TO ARRAY[1..4] OF BYTE;
END_VAR
VAR
END_VAR
pOut^[1]:=pIn^[4];
pOut^[2]:=pIn^[3];
pOut^[3]:=pIn^[2];
pOut^[4]:=pIn^[1];
END_FUNCTION

(* POU Utils Functions/CHKSTRING, ST *)
FUNCTION CHKSTRING : BOOL
VAR_INPUT
	pString: POINTER TO BYTE;
	pPattern: POINTER TO BYTE;
END_VAR
VAR
END_VAR
CHKSTRING:=TRUE;
WHILE pPattern^<>0 AND CHKSTRING DO
	IF pPattern^<>pString^ THEN CHKSTRING:=FALSE; END_IF
	pString:=pString+1;
	pPattern:=pPattern+1;
END_WHILE
END_FUNCTION

(* POU TCP_Remote/Remote_Proc, ST *)
PROGRAM Remote_Proc
VAR
	s1:         	TCPSERVER;
	Enable: 		BOOL;
	Connected: 		BOOL;
	Error: 			DINT;

	TxData:			ARRAY [0..MAX_SEND_TCP_SERVER] OF BYTE;
	TxLen:			DINT;
	TxTrig:			BOOL;

	RxData:			ARRAY [0..MAX_RECEIVE_TCP_SERVER] OF BYTE;
	RxLen:			DINT;

	Status:			DINT;

	(* Command interpreter *)

	Cmd_Buf:		ARRAY [0..MAX_RECEIVE_TCP_SERVER] OF BYTE;
	Cmd_Buf_U16:	POINTER TO WORD;
	Cmd_Buf_INT:	POINTER TO INT;
	Cmd_BufLen:		WORD;
	Cmd_St:			WORD;

	Cmd_Obj:		WORD;
	Cmd_ObjIdx:		WORD;
	Cmd_C:			WORD;
	Cmd_R:			WORD;
	Cmd_CLen:		WORD;
	Cmd_RLen:		WORD;

	i : WORD;
	j : INT;

END_VAR
(*=== State machine ===*)
CASE Status OF
	0: (* Startup *)
		TxLen:=0; TxTrig:=FALSE;
		RxLen:=0;
		Enable:=TRUE;
		Status:=1;

	1: (* Wait incoming connection *)
		IF Connected THEN
			(* Log access *)
			LogEv(EL_Log,EO_VPN,1,5,'Remote');
			(* Send welcome message *)
			ADDSTRING(pTxData:=ADR(TxData), pString:=ADR(Remote_WELCOME), TxLen:=TxLen);
			TxTrig:=TRUE;
			Cmd_BufLen:=0;
			Cmd_St:=0;
			Status:=2;
		END_IF
		IF Error>1 THEN
			Enable:=FALSE;
			Status:=0;
		END_IF

	2: (* Wait command *)
		IF RxLen>0 THEN
			(*=== Interpreter start ===*)
			IF Cmd_BufLen+(RxLen/2)>=MAX_RECEIVE_TCP_SERVER THEN
				(* ERROR *)
				Cmd_BufLen:=0;
			ELSE
				i:=HEXTORAW(pString:=ADR(RxData), StringLen:=DINT_TO_WORD(RxLen), pData:=ADR(Cmd_Buf[Cmd_BufLen]));
				Cmd_BufLen:=Cmd_BufLen+i;
			END_IF
			IF Cmd_BufLen>=8 THEN
				Cmd_Buf_U16:=ADR(Cmd_Buf[6]);
				IF Cmd_BufLen>=(8+Cmd_Buf_U16^) THEN
					Cmd_CLen:=Cmd_Buf_U16^;
					Cmd_Buf_U16:=ADR(Cmd_Buf[0]); Cmd_Obj:=Cmd_Buf_U16^;
					Cmd_Buf_U16:=ADR(Cmd_Buf[2]); Cmd_ObjIdx:=Cmd_Buf_U16^;
					Cmd_Buf_U16:=ADR(Cmd_Buf[4]); Cmd_C:=Cmd_Buf_U16^;
					Command();
					Cmd_BufLen:=0;
				END_IF
			END_IF
			(*=== Interpreter end ===*)
			RxLen:=0;
		END_IF
		IF NOT Connected THEN
			Status:=0;
		END_IF

ELSE
	Status:=0;
END_CASE


(*=== Execute server lib ===*)
s1(
	xEnable				:= Enable,
	wPortNumber			:= Remote_PORT,
	tServerTimeOut		:= t#15m,
	ptSendData			:= ADR(TxData),
	diSendCount			:= TxLen,
	xStartSend			:= TxTrig,
	aReceiveBuffer		:= RxData,
	diReceiveCount		:= RxLen,
	xClientConnected	=> Connected,
	diError				=> Error
);
END_PROGRAM
ACTION Cmd_CAL:
(* Check index *)(*
IF Cmd_ObjIdx<1 OR Cmd_ObjIdx>2 THEN
	Cmd_R:=2;
	RETURN;
END_IF

(* Process command *)
CASE Cmd_C OF

	3: (* TRY REARM *)
		IF Cmd_ObjIdx=1 THEN
			CAL01.Rearm:=TRUE;
		ELSE
			CAL02.Rearm:=TRUE;
		END_IF

ELSE
	Cmd_R:=3;
END_CASE
*);
END_ACTION
ACTION Cmd_CRON:
(* Check index *)(*
IF Cmd_ObjIdx<1 OR Cmd_Obj=2 OR Cmd_ObjIdx>6 THEN
	Cmd_R:=2;
	RETURN;
END_IF

(* Process command *)
CASE Cmd_C OF

	1: (* GET PROFILE *)
		IF Cmd_CLen<>3 THEN
			Cmd_R:=4;
		ELSE
			(* Load profile *)
			CronEd.CN_Sel:=WORD_TO_BYTE(Cmd_ObjIdx);
			Cmd_Buf_U16:=ADR(Cmd_Buf[8]);
			CronEd.CN_YSel:=Cmd_Buf_U16^;
			CronEd.PR_Sel:=Cmd_Buf[10];
			CronEd.PR_Load_Exe();
			(* Copy data *)
			Cmd_RLen:=192;
			TxLen:=TxLen+RAWTOHEX(ADR(CronEd.PR.Setpoint),192,ADR(TxData[TxLen]));
		END_IF

	2: (* SET PROFILE *)
		IF Cmd_CLen<>(3+192) THEN
			Cmd_R:=4;
		ELSE
			(* Save profile *)
			CronEd.CN_Sel:=WORD_TO_BYTE(Cmd_ObjIdx);
			Cmd_Buf_U16:=ADR(Cmd_Buf[8]);
			CronEd.CN_YSel:=Cmd_Buf_U16^;
			CronEd.PR_Sel:=Cmd_Buf[10];
			MEMCPY(ADR(Cmd_Buf[11]),ADR(CronEd.PR.Setpoint),192);
			CronEd.PR_Save_Exe();
		END_IF

	5: (* GET CALENDAR MONTH *)
		IF Cmd_CLen<>3 THEN
			Cmd_R:=4;
		ELSE
			(* Load calendar *)
			CronEd.CN_Sel:=WORD_TO_BYTE(Cmd_ObjIdx);
			Cmd_Buf_U16:=ADR(Cmd_Buf[8]);
			CronEd.CN_YSel:=Cmd_Buf_U16^;
			CronEd.CA_Sel:=Cmd_Buf[10];
			CronEd.CA_Load_Exe();
			(* Copy data *)
			Cmd_RLen:=32;
			TxLen:=TxLen+RAWTOHEX(ADR(CronEd.CA.Profile),32,ADR(TxData[TxLen]));
		END_IF

	6: (* SET CALENDAR MONTH *)
		IF Cmd_CLen<>(3+32) THEN
			Cmd_R:=4;
		ELSE
			(* Save calendar *)
			CronEd.CN_Sel:=WORD_TO_BYTE(Cmd_ObjIdx);
			Cmd_Buf_U16:=ADR(Cmd_Buf[8]);
			CronEd.CN_YSel:=Cmd_Buf_U16^;
			CronEd.CA_Sel:=Cmd_Buf[10];
			MEMCPY(ADR(Cmd_Buf[11]),ADR(CronEd.CA.Profile),32);
			CronEd.CA_Save_Exe();
		END_IF

ELSE
	Cmd_R:=3;
END_CASE
*);
END_ACTION
ACTION Cmd_GRU:
(* Check index *)(*
IF Cmd_ObjIdx<>1 THEN
	Cmd_R:=2;
	RETURN;
END_IF

(* Process command *)
CASE Cmd_C OF

	1: (* GET CLIMATIC *)
		Cmd_RLen:=20;
		FOR i:=0 TO 4 DO
			j:=DINT_TO_INT(GRU01_Clima.Points[i].X);
			TxLen:=TxLen+RAWTOHEX(ADR(j),2,ADR(TxData[TxLen]));
			j:=DINT_TO_INT(GRU01_Clima.Points[i].Y);
			TxLen:=TxLen+RAWTOHEX(ADR(j),2,ADR(TxData[TxLen]));
		END_FOR

	2: (* SET CLIMATIC *)
		IF Cmd_CLen<>20 THEN
			Cmd_R:=4;
		ELSE
			FOR i:=0 TO 4 DO
				Cmd_Buf_INT:=ADR(Cmd_Buf[8+4*i]); j:=Cmd_Buf_INT^;
				GRU01_Clima.Points[i].X:=INT_TO_DINT(j);
				Cmd_Buf_INT:=ADR(Cmd_Buf[10+4*i]); j:=Cmd_Buf_INT^;
				GRU01_Clima.Points[i].Y:=INT_TO_DINT(j);
			END_FOR
		END_IF

ELSE
	Cmd_R:=3;
END_CASE
*);
END_ACTION
ACTION Cmd_PDC:
;(* Check index *)(*
IF Cmd_ObjIdx<>1 THEN
	Cmd_R:=2;
	RETURN;
END_IF

(* Process command *)
CASE Cmd_C OF

	3: (* TRY REARM *)
		PDC01.Rearm:=TRUE;

ELSE
	Cmd_R:=3;
END_CASE
*);
END_ACTION
ACTION Cmd_SYS:
(* Check index *)
IF Cmd_ObjIdx<>0 THEN
	Cmd_R:=2;
	RETURN;
END_IF

(* Process command *)
CASE Cmd_C OF

	0: (* ECHO *)
		IF Cmd_CLen<>0 THEN
			TxLen:=0;
		END_IF

	1: (* LOG REQUEST *)
		LogTrig();

	2: (* REARM *)
		Sys.Warning:=FALSE;
		Sys.Alarm:=FALSE;
		Sys.AlarmStop:=FALSE;

	3: (* GET INFO1 *)
		Cmd_RLen:=6;
		TxLen:=TxLen+RAWTOHEX(ADR(Plant_SN),4,ADR(TxData[TxLen]));
		TxLen:=TxLen+RAWTOHEX(ADR(Plant_SW_VER),2,ADR(TxData[TxLen]));

ELSE
	Cmd_R:=3;
END_CASE
END_ACTION
ACTION Command:
(* Default response OK/NODATA *)
Cmd_R:=0;
Cmd_RLen:=0;
TxLen:=16;

(* Check object *)
CASE Cmd_Obj OF

	EO_SYS:
		Cmd_SYS();
(*
	EO_GRU:
		Cmd_GRU();

	EO_PDC:
		Cmd_PDC();

	EO_CAL:
		Cmd_CAL();

	EO_CRON:
		Cmd_CRON();
*)
ELSE
	Cmd_R:=1;
END_CASE

(* Generate response *)
IF TxLen>0 THEN
	RAWTOHEX(ADR(Cmd_Obj)	,2,ADR(TxData[ 0]));
	RAWTOHEX(ADR(Cmd_ObjIdx),2,ADR(TxData[ 4]));
	RAWTOHEX(ADR(Cmd_R)		,2,ADR(TxData[ 8]));
	RAWTOHEX(ADR(Cmd_RLen)	,2,ADR(TxData[12]));
	TxTrig:=TRUE;
END_IF
END_ACTION

(* POU Utils Functions/TCPSERVER, ST *)
FUNCTION_BLOCK TCPSERVER
(***********************************************************************************************************	*)
(* Version: 1.6                                    			          											*)
(* Date: 11.02.2011                                   					          							    *)
(***********************************************************************************************************	*)
(* WAGO Kontakttechnik GmbH Hansastr. 27 32423 Minden(Westf.)													*)
(* Tel. +0049 571/887-0 Fax. +0049 571/887-0																	*)
(* Author: VB																									*)
(***********************************************************************************************************	*)
(*Description:	A TCP server to read and write data													       		*)
(*Historie:																										*)
(*Version 1.6: 11.02.2011: Changes according to 750-880/881											 			*)
(*Version 1.5: 27.11.2008 Bugfix allow reuse port																*)
(*Version 1.4: 13.10.2008 Bugfix transmitting large data														*)
(*Version 1.3: 15.01.2007 Changes according to FW11																*)
(*Version 1.2: 09.03.2006 Changes for socket handle 0											       			*)
(*Version 1.1: 14.02.2005 Release																				*)
(***********************************************************************************************************	*)
VAR CONSTANT
	STATE_INIT     				 : BYTE:= 0;
	STATE_OPEN     				 : BYTE:= 1;
	STATE_TX       				 : BYTE:= 20;
	STATE_RX       				 : BYTE:= 30;
	STATE_CLOSE    				 : BYTE:= 40;
	STATE_ERROR_TRAP		 	 : BYTE:= 200;
END_VAR
VAR_INPUT
	xEnable    					: BOOL;	 (* Set TRUE to enable function block *)
	wPortNumber					: WORD;  (* Port *)
	tServerTimeOut				: TIME:=t#50s;
	ptSendData					: POINTER TO ARRAY[0..MAX_SEND_TCP_SERVER] OF BYTE;
	diSendCount					: DINT;
END_VAR
VAR_OUTPUT
	xClientConnected  			: BOOL:= FALSE;
	diError 					: DINT:= 0;
END_VAR
(* Status Codes -----------------------------------------
	16#8001 => No socket descriptor available 
	16#8002 => SysSockBind fails 
	16#8003 => SysSockListen fails 
	16#8004 => switching to none blocking mode fails
	16#8005 => SysSockClose() returns FALSE 
    16#8006 => SysSockConnect() fails
    16#8007 => SysSockSend() fails
	16#8008 => error state machine 
	16#8009 => timeout while waiting for data from server 
	16#0001 => server waiting for client to establish connection
------------------------------------------------------------*)
VAR_IN_OUT
	xStartSend					: BOOL;
	aReceiveBuffer				: ARRAY [0..MAX_RECEIVE_TCP_SERVER] OF BYTE;
	diReceiveCount				: DINT;
END_VAR

VAR
	m_State    					: BYTE:= 0;
	m_ReceiveBuffer				: ARRAY [0..MAX_RECEIVE_TCP_SERVER_SOCKET] OF BYTE;
	m_ServerSocket				: DINT:= SOCKET_INVALID;
	m_Socket					: DINT:= SOCKET_INVALID;
	m_AddressInfo				: SOCKADDRESS;
	m_BytesReceived				: DINT;
	m_diReturn					: DINT;
	m_xReturn					: BOOL;
	m_SizeSockadr				: DWORD;
	m_ConnectionWatchdog		: TON;
	m_Flags						: DINT;
	m_NoneBlocking   			: DINT:= 1;
	m_Blocking   				: DINT:= 0;
	i							: INT;
	m_count						: DINT;
	diOption					: DINT := 1;
	on: DINT;
END_VAR
IF xEnable THEN
	CASE m_State OF
		STATE_INIT:
			(* Create Socket *)
			m_ServerSocket:= SysSockCreate( SOCKET_AF_INET, SOCKET_STREAM, 0);
			IF m_ServerSocket = SOCKET_INVALID THEN
				(* *)
				diError:= 16#8001;
				m_State:= STATE_ERROR_TRAP;
				RETURN;
			ELSE
				;
			END_IF
			(* Address bindings *)
			(********************)
			on:=1;
			SysSockSetOption( m_ServerSocket, SOCKET_SOL, SOCKET_SO_REUSEADDR, ADR(on), SIZEOF(on) );

			m_AddressInfo.sin_family:= SOCKET_AF_INET;
			m_AddressInfo.sin_port  := SysSockHtons( wPortNumber);
			m_AddressInfo.sin_addr  := SOCKET_INADDR_ANY;
			IF NOT SysSockBind( m_ServerSocket, ADR(m_AddressInfo), SIZEOF(m_AddressInfo)) THEN
				diError:= 16#8002;
				m_State:= STATE_ERROR_TRAP;
				RETURN;
			END_IF
			(* Wait for connections *)
			(************************)
			IF NOT SysSockListen( m_ServerSocket, 1) THEN
				diError:= 16#8003;
				m_State:= STATE_ERROR_TRAP;
			END_IF

			(* Puts SOCKET in NonBlocking mode *)
			m_diReturn:= SysSockIoctl( m_ServerSocket, SOCKET_FIONBIO, ADR(m_NoneBlocking));

			m_State:= STATE_OPEN;


		STATE_OPEN: 	(* Waiting for incomming connection *)
				m_SizeSockadr:=SIZEOF(m_AddressInfo);
				m_Socket:= SysSockAccept( m_ServerSocket, ADR(m_AddressInfo), ADR(m_SizeSockadr));
				diError:=State_open;
				IF m_Socket <> SOCKET_INVALID THEN
					xClientConnected:=TRUE;
					(*Set Push-Bit:new V1.5*)
					IF ADR(%MW0)=16#30000000  OR ADR(%MW0)=16#20000000 THEN (*841 or 881*)
						SysSockSetOption(
							diSocket:=m_Socket,
							diLevel:=6,
							diOption:=SOCKET_TCP_NODELAY,
							pOptionValue:=ADR(diOption),
							diOptionLength:=SIZEOF(diOption));
					ELSE
							;
					END_IF
					SysSockIoctl( m_Socket, SOCKET_FIONBIO, ADR(m_NoneBlocking));
					m_State:= STATE_RX;
					diError:=0;
				END_IF

		STATE_RX:
					m_BytesReceived:= SysSockRecv( m_Socket, ADR(m_ReceiveBuffer), SIZEOF(m_ReceiveBuffer), 0);
					CASE m_BytesReceived OF
					-1:(*no data available or error occured*)
						m_ConnectionWatchdog(IN:=TRUE , PT:=tServerTimeOut );
						IF m_connectionWatchdog.Q THEN
							m_State:= STATE_CLOSE;
							m_ConnectionWatchdog(IN:=FALSE);(*reset connection watchdog*)
							diError := 16#8009;
						END_IF
					0:(* socket was "gracefully closed"  *)
						m_State:= STATE_CLOSE;
						diError := 16#8003;
					ELSE
						(* Copy received data into receive buffer *)
						(********************************)
						FOR i:= 0 TO DINT_TO_INT(m_BytesReceived	)-1 DO
							aReceiveBuffer[diReceiveCount]:= m_ReceiveBuffer[i];
							diReceiveCount:=(diReceiveCount+1) MOD SIZEOF(aReceiveBuffer);
						END_FOR

						m_ConnectionWatchdog(IN:=FALSE);(*reset connection watchdog*)
					END_CASE

				(*send data*)
				IF xStartSend	 THEN
					m_State := STATE_TX;
				END_IF

	STATE_TX:	 (* send TCP-message *)
		m_diReturn := SysSockSend(diSocket := m_Socket,
								  pbyBuffer := ADR(ptSendData^[m_count]),(*geändert V1.4 bisher: [0] *)
								  diBufferSize := diSendCount-m_count,
								  diFlags :=m_Flags);
		CASE m_diReturn OF
		-1:	(* ERROR or data could not yet be send (V1.3 due to new FW11) *)
			m_ConnectionWatchdog(IN:=TRUE , PT:=tServerTimeOut );
			IF m_connectionWatchdog.Q THEN
				m_State:= STATE_CLOSE;
				m_ConnectionWatchdog(IN:=FALSE);(*reset connection watchdog*)
				diError := 16#8007;
			END_IF
		0: (* socket was "gracefully closed"  *)
			m_State := STATE_CLOSE;
			diError := 16#8003;
		ELSE (* succesful *)
			m_count:=m_count+m_diReturn;
			IF m_count>=diSendCount THEN
				diError := 16#0000;
				m_State := STATE_RX;
				m_count:=0;
				xStartSend:=FALSE;
			END_IF
			m_ConnectionWatchdog(IN:=FALSE);(*reset connection watchdog*)
		END_CASE


		STATE_CLOSE:	(* Close the server *)

		IF ADR(%MW0)=16#30000000  OR ADR(%MW0)=16#20000000 THEN (*841 or 881*)
			;
		ELSE
			IF m_Socket>=0 THEN
				SysSockShutdown(m_Socket, 0);;(*870*)
			END_IF
		END_IF
		IF m_Socket>=0 THEN
			SysSockClose( m_Socket);
		END_IF
		xClientConnected:= FALSE;
		m_State:= STATE_OPEN; (* Try to open the server again *)
		m_ConnectionWatchdog(IN:=FALSE);(*reset connection watchdog*)

		STATE_ERROR_TRAP: (* Error Read/Write socket  *)
			m_State:= STATE_ERROR_TRAP;

	ELSE  (* Bad FSM code trap  *)
			m_State:= STATE_ERROR_TRAP;
			diError:= 16#8008;
	END_CASE;
ELSE
	IF m_State <> STATE_INIT THEN
		IF ADR(%MW0)=16#30000000  OR ADR(%MW0)=16#20000000 THEN (*841 or 881*)
			;
		ELSE
			IF m_Socket>=0 THEN
				SysSockShutdown(m_Socket, 0);;(*870*)
			END_IF
		END_IF
		IF m_Socket>=0 THEN
			SysSockClose( m_Socket);
		END_IF
		IF ADR(%MW0)=16#30000000  OR ADR(%MW0)=16#20000000 THEN (*841 or 881*)
			;
		ELSE
			IF m_ServerSocket>=0 THEN
				SysSockShutdown(m_ServerSocket, 0);;(*870*)
			END_IF
		END_IF
		IF m_ServerSocket>=0 THEN
			SysSockClose( m_ServerSocket);
		END_IF
		xClientConnected:= FALSE;
		diError:= 0;
		m_State:= STATE_init; (* Try to open the server again *)
		m_ConnectionWatchdog(IN:=FALSE);(*reset connection watchdog*)
	END_IF
END_IF
END_FUNCTION_BLOCK

(* POU TCP_Logger/LogEv, ST *)
FUNCTION LogEv : BOOL
VAR_INPUT
	Level	: en_Logger_ErrLev;
	Object  : en_SYS_Objects;
	Index	: WORD;
	Error	: WORD;
	Message : STRING;
END_VAR
VAR
	s1 : STRING(160);
	i  : INT;
END_VAR
(* Execute error level operations *)
CASE Level OF
	EL_Wrn: 		Sys.Warning:=TRUE;
	EL_Alarm: 		Sys.Alarm:=TRUE;
	EL_AlarmStop: 	Sys.Alarm:=TRUE; (* GO TO STOP STATE!! *)
END_CASE

(* Fill lastlog list *)
s1:=CONCAT(Sys.Time_LogString,';Lev=');
s1:=CONCAT(s1,INT_TO_STRING(Level));
s1:=CONCAT(s1,';Obj=');
s1:=CONCAT(s1,INT_TO_STRING(Object));
s1:=CONCAT(s1,';Idx=');
s1:=CONCAT(s1,WORD_TO_STRING(Index));
s1:=CONCAT(s1,';Err=');
s1:=CONCAT(s1,WORD_TO_STRING(Error));
Sys.LastLogs_Dat[Sys.LastLogs_Idx]:=s1;
Sys.LastLogs_Msg[Sys.LastLogs_Idx]:=Message;
Sys.LastLogs_Idx:=Sys.LastLogs_Idx+1;
IF Sys.LastLogs_Idx>5 THEN Sys.LastLogs_Idx:=0; END_IF

(*---------------------------------------------------------------*)
(*---------------------------------------------------------------*)
Logger.TLen:=0;
(* Set GET header *)
ADDSTRING(ADR(Logger.TData), ADR(Logger_GETSTART), Logger.TLen);

(* Insert Header *)
s1:=INSERT('ID=&V=1&D=',DWORD_TO_STRING(Plant_SN),3);
s1:=CONCAT(s1,Sys.Time_LogString);
s1:=CONCAT(s1,'&S=');
IF Sys.Alarm THEN i:=2; ELSIF Sys.Warning THEN i:=1; ELSE i:=0; END_IF
s1:=CONCAT(s1,INT_TO_STRING(i));
ADDSTRING(ADR(Logger.TData), ADR(s1), Logger.TLen);

(* Insert ERR *)
s1:=CONCAT('&ERR=',INT_TO_STRING(Level));
s1:=CONCAT(s1,';');
s1:=CONCAT(s1,INT_TO_STRING(Object));
s1:=CONCAT(s1,';');
s1:=CONCAT(s1,WORD_TO_STRING(Index));
s1:=CONCAT(s1,';');
s1:=CONCAT(s1,WORD_TO_STRING(Error));
s1:=CONCAT(s1,';');
ADDSTRING(ADR(Logger.TData), ADR(s1), Logger.TLen);
s1:=Message;
STR_NOSPACES(ADR(s1));
ADDSTRING(ADR(Logger.TData), ADR(s1), Logger.TLen);

(* Finalize string *)
ADDSTRING(ADR(Logger.TData), ADR(Logger_GETEND), Logger.TLen);

(*---------------------------------------------------------------*)
(*---------------------------------------------------------------*)

Logger_Send();
END_FUNCTION

(* POU Utils Functions/ADDSTRING, ST *)
FUNCTION ADDSTRING : BOOL (* Append string to a byte buffer *)
VAR_INPUT
	pTxData: POINTER TO BYTE;
	pString: POINTER TO BYTE;
END_VAR
VAR_IN_OUT
	TxLen: DINT;
END_VAR
VAR
END_VAR
pTxData:=pTxData+TxLen;
WHILE pString^<>0 DO
	pTxData^:=pString^;
	pString:=pString+1;
	pTxData:=pTxData+1;
	TxLen:=TxLen+1;
END_WHILE
END_FUNCTION

(* POU Utils Functions/STR_NOSPACES, ST *)
FUNCTION STR_NOSPACES : BOOL (* Replace spaces and bad chars with allowed ones, used as HTTP-GET validator *)
VAR_INPUT
	pString: POINTER TO BYTE;
END_VAR
VAR
END_VAR
WHILE pString^<>0 DO
	IF pString^=16#20 (* space *) THEN pString^:=16#5F; (*'_'*) END_IF
	pString:=pString+1;
END_WHILE
END_FUNCTION

(* POU TCP_Logger/Logger_Send, ST *)
FUNCTION Logger_Send : BOOL
VAR
	hFile: 	DWORD;
	pos:	DWORD;
END_VAR
(* Read log position *)
pos:=SysFileGetSize(Logger_DataFile);
(* Check log size, bckup and erase if no pending messages *)
IF pos>100000000 (*100M*) THEN
	hFile:=SysFileOpen(Logger_IndexFile,'r');
	IF hFile=0 THEN
		SysFileDelete(Logger_DataFileOld);
		SysFileRename(Logger_DataFile,Logger_DataFileOld);
		pos:=0;
	ELSE
		SysFileClose(hFile);
	END_IF
END_IF
(* Write message on log file *)
hFile:=SysFileOpen(Logger_DataFile,'a');
IF hFile<>0 THEN
	SysFileWrite(hFile, ADR(Logger.TData), Logger.TLen);
	SysFileClose(hFile);
ELSE
	Sys.Warning:=TRUE;
END_IF


(* Check logger status *)
IF Logger.SendReq=FALSE THEN
	(* Set log position for recovery *)
	Logger.SendIdx:=pos;
	(* Copy message data *)
	MEMCPY(ADR(Logger.TData),ADR(Logger.SendData),DINT_TO_WORD(Logger.TLen));
	Logger.SendLen:=Logger.TLen;
	(* Trigger request *)
	Logger.SendReq:=TRUE;
ELSE
	(* Add message position+size in recovery indexes *)
	hFile:=SysFileOpen(Logger_IndexFile,'a');
	SysFileWrite(hFile, ADR(pos), SIZEOF(pos));
	SysFileWrite(hFile, ADR(Logger.TLen), SIZEOF(Logger.TLen));
	SysFileClose(hFile);
END_IF
END_FUNCTION

(* POU Utils Functions/MEMCPY, ST *)
FUNCTION MEMCPY:BOOL
VAR_INPUT
	pSourceAddress:POINTER TO ARRAY[1..2] OF BYTE;
	pDestinationAddress:POINTER TO ARRAY[1..2] OF BYTE;
	BytesToCopy:WORD;
END_VAR
VAR
END_VAR
WHILE (BytesToCopy > 0) DO
	pDestinationAddress^[1]:=pSourceAddress^[1]; (* copy bytes from source to destination *)
	pDestinationAddress:=ADR(pDestinationAddress^[2]); (* increment destination *)
	pSourceAddress:=ADR(pSourceAddress^[2]);(* increment source *)
	BytesToCopy:=BytesToCopy -1; (* decrement number of bytes to copy *)
END_WHILE
END_FUNCTION

(* POU Utils Functions/HEXTORAW, ST *)
FUNCTION HEXTORAW : WORD
VAR_INPUT
	pString		: POINTER TO BYTE;
	StringLen	: WORD;
	pData		: POINTER TO BYTE;
END_VAR
VAR
	xl: WORD;
	xi: WORD;
	xr: BYTE;
END_VAR
xl:=0;
xi:=0;

WHILE xi<StringLen DO

	IF pString^>=97 AND pString^<=102 THEN
		xr := pString^ - 87;
	ELSIF pString^>=65 AND pString^<=70 THEN
		xr := pString^ - 55;
	ELSIF pString^>=48 AND pString^<=57 THEN
		xr := pString^ - 48;
	ELSE
		xr := 16;
	END_IF

	IF xr<16 THEN
		IF (xi AND 1)=0 THEN
			pData^ := xr * 16;
		ELSE
			pData^ := pData^ + xr;
			pData := pData + 1;
			xl := xl + 1;
		END_IF
	END_IF

	xi := xi + 1;
	pString := pString + 1;

END_WHILE

HEXTORAW:=xl;
END_FUNCTION

(* POU Utils Functions/RAWTOHEX, ST *)
FUNCTION RAWTOHEX : WORD
VAR_INPUT
	pData: POINTER TO BYTE;
	DataLen: WORD;
	pString: POINTER TO BYTE;
END_VAR
VAR
	xl: WORD;
END_VAR
xl:=0;

WHILE DataLen>0 DO

	pString^ := (pData^ / 16#10) + 48 + (((pData^ / 16#10)/10)*7);
	pString:=pString+1;
	pString^ := (pData^ AND 16#0F)  + 48 + (((pData^ AND 16#0F)/10)*7);
	pString:=pString+1;
	pData:=pData+1;
	DataLen:=DataLen-1;
	xl:=xl+2;

END_WHILE

(*pString^:=0;*)

RAWTOHEX:=xl;
END_FUNCTION

(* POU Utils/USRLED_Update, ST *)
PROGRAM USRLED_Update
VAR
	OldStatus: en_SYS_Status;

	aFS : ARRAY [0..24] OF FLASHING_SEQUENCE :=
		(Colour:=GREEN,  Frequency:=1,   Relation:=128, Duration:=t#0s,    NextIndex:=0),  (* 0 => RUNNING *)
		(Colour:=ORANGE, Frequency:=1,   Relation:=128, Duration:=t#0s,    NextIndex:=1),  (* 1 => INIT *)
		(Colour:=RED,    Frequency:=4,   Relation:=128, Duration:=t#0s,    NextIndex:=2),  (* 2 => ERROR *)
		(Colour:=RED,    Frequency:=10,  Relation:=128, Duration:=t#0s,    NextIndex:=3),  (* 3 => ALARM *)
		(Colour:=ORANGE, Frequency:=200, Relation:=16,  Duration:=t#100ms, NextIndex:=11), (* 10 *)
		(Colour:=ORANGE, Frequency:=200, Relation:=32,  Duration:=t#100ms, NextIndex:=12),
		(Colour:=ORANGE, Frequency:=200, Relation:=64,  Duration:=t#100ms, NextIndex:=13),
		(Colour:=ORANGE, Frequency:=200, Relation:=128, Duration:=t#100ms, NextIndex:=14),
		(Colour:=ORANGE, Frequency:=200, Relation:=192, Duration:=t#100ms, NextIndex:=15),
		(Colour:=ORANGE, Frequency:=200, Relation:=128, Duration:=t#100ms, NextIndex:=16),
		(Colour:=ORANGE, Frequency:=200, Relation:=64,  Duration:=t#100ms, NextIndex:=17),
		(Colour:=ORANGE, Frequency:=200, Relation:=32,  Duration:=t#100ms, NextIndex:=18),
		(Colour:=ORANGE, Frequency:=200, Relation:=16,  Duration:=t#100ms, NextIndex:=19),
		(Colour:=ORANGE, Frequency:=200, Relation:=8,   Duration:=t#100ms, NextIndex:=10),
		(Colour:=GREEN,  Frequency:=200, Relation:=16,  Duration:=t#100ms, NextIndex:=21), (* 20 *)
		(Colour:=GREEN,  Frequency:=200, Relation:=32,  Duration:=t#100ms, NextIndex:=22),
		(Colour:=GREEN,  Frequency:=200, Relation:=64,  Duration:=t#100ms, NextIndex:=23),
		(Colour:=GREEN,  Frequency:=200, Relation:=128, Duration:=t#100ms, NextIndex:=24),
		(Colour:=GREEN,  Frequency:=200, Relation:=192, Duration:=t#100ms, NextIndex:=25),
		(Colour:=GREEN,  Frequency:=200, Relation:=128, Duration:=t#100ms, NextIndex:=26),
		(Colour:=GREEN,  Frequency:=200, Relation:=64,  Duration:=t#100ms, NextIndex:=27),
		(Colour:=GREEN,  Frequency:=200, Relation:=32,  Duration:=t#100ms, NextIndex:=28),
		(Colour:=GREEN,  Frequency:=200, Relation:=16,  Duration:=t#100ms, NextIndex:=29),
		(Colour:=GREEN,  Frequency:=200, Relation:=8,   Duration:=t#100ms, NextIndex:=20);

	pFS : POINTER TO FLASHING_SEQUENCE;


END_VAR
IF Sys.Status <> OldStatus THEN

	OldStatus:=Sys.Status;

	CASE OldStatus OF

		S_STARTUP:
			pFS:=ADR(aFS);
			SET_FLASHING_SEQUENCE(EN:=TRUE, POINTER_TO_POINTER_TO_ARRAY:=ADR(pFS));
			SET_FLASHING_SEQUENCE_INDEX(EN:=TRUE, IMMEDIATE:=FALSE, INDEX:=1);
			START_FLASHING_SEQUENCE(EN:=TRUE);

		S_RUNNING:
			SET_FLASHING_SEQUENCE_INDEX(EN:=TRUE, IMMEDIATE:=TRUE, INDEX:=0);

	END_CASE

END_IF
END_PROGRAM

(* POU Utils/CSV_Log, ST *)
FUNCTION CSV_Log : BOOL
VAR_INPUT
END_VAR
VAR CONSTANT
	LogFileName:STRING:='S:\LOGS_ID4V3.CSV';
END_VAR
VAR
	s1 : STRING(256);
	hFile: 	DWORD;
END_VAR
(* Check file presence *)
hFile:=SysFileOpen(LogFileName,'r');
IF hFile=0 THEN
	(*** File not exist *** Create file and write header *)
	hFile:=SysFileOpen(LogFileName,'w');
	IF hFile<>0 THEN
		(* Write CSV header *)
		s1:='DATE-TIME;T-Amb;T-GRU01-SetP;T-GRU01-Send;T-GRU01-Ret;T-GRU01-Amb;T_S01;T_S02;F-PDC01-Flow;T-PDC01-Send;T-PDC01-Ret;';
		SysFileWrite(hFile, ADR(s1), LEN(s1));
		s1:='T-CTB01-Send;T-CTB01-Ret;F-CTB01-Flow;P-CTB01-Power;E-CTB01-Energy';
		SysFileWrite(hFile, ADR(s1), LEN(s1));
		SysFileWrite(hFile, ADR(Logger_CRLF), LEN(Logger_CRLF));
	END_IF
ELSE
	(*** File exist *** Close file and reopen in append mode *)
	SysFileClose(hFile);
	hFile:=SysFileOpen(LogFileName,'a');
END_IF

(* Log to file *)
IF hFile<>0 THEN
	(* Date stamp *)
	s1:=REPLACE( Sys.Time_LogString , ' ' , 1 , 11 );
	SysFileWrite(hFile, ADR(s1), LEN(s1));
	(* Log data 1 *)
	s1:=CONCAT(';', INT_TO_STRING(T_AMB) );
	s1:=CONCAT(s1 , ';');
	s1:=CONCAT(s1 , INT_TO_STRING(GRU01.ActSetPoint) );
	s1:=CONCAT(s1 , ';');
	s1:=CONCAT(s1 , INT_TO_STRING(GRU01.TSend) );
	s1:=CONCAT(s1 , ';');
	s1:=CONCAT(s1 , INT_TO_STRING(GRU01.TRet) );
	s1:=CONCAT(s1 , ';');
	s1:=CONCAT(s1 , INT_TO_STRING(GRU01.TAmb) );
	s1:=CONCAT(s1 , ';');
	s1:=CONCAT(s1 , INT_TO_STRING(T_S01) );
	s1:=CONCAT(s1 , ';' );
	s1:=CONCAT(s1 , INT_TO_STRING(T_S02) );
	s1:=CONCAT(s1 , ';' );
	s1:=CONCAT(s1 , WORD_TO_STRING(PDC01.Flow) );
	s1:=CONCAT(s1 , ';' );
	s1:=CONCAT(s1 , INT_TO_STRING(PDC01.TSend) );
	s1:=CONCAT(s1 , ';');
	s1:=CONCAT(s1 , INT_TO_STRING(PDC01.TRet) );
	SysFileWrite(hFile, ADR(s1), LEN(s1));
	(* Log data 2 *)
	s1:=CONCAT(';', CTB01.M1.utFTemp.Value );
	s1:=CONCAT(s1 , ';');
	s1:=CONCAT(s1 , CTB01.M1.utRTemp.Value );
	s1:=CONCAT(s1 , ';');
	s1:=CONCAT(s1 , CTB01.M1.utFlow.Value );
	s1:=CONCAT(s1 , ';');
	s1:=CONCAT(s1 , CTB01.M1.utPower.Value );
	s1:=CONCAT(s1 , ';');
	s1:=CONCAT(s1 , CTB01.M1.utEnergy.Value );
	SysFileWrite(hFile, ADR(s1), LEN(s1));
	(* Add line CRLF and close *)
	SysFileWrite(hFile, ADR(Logger_CRLF), LEN(Logger_CRLF));
	SysFileClose(hFile);
END_IF
END_FUNCTION

(* POU Plant/SYS_Proc, ST *)
PROGRAM SYS_Proc
VAR
(*	fALARM_PB		:FLT_TAP;
	fALARM_TB		:FLT_TAP;
	fALARM_PM		:FLT_TAP; *)

(*	fGZB_ST			:FLT_TAP; (* GATEWAY ZIGBEE *)*)
(*	fVPN_OUT1		:FLT_TAP; (* VPN - CONNECT *)*)
	fVPN_OUT2		:FLT_TAP; (* VPN - STATUS *)
(*	fKEY_CT_ST		:FLT_TAP; (* DOOR01 - Porta primaria *)*)
(*	fKEY_SCT_ST		:FLT_TAP; (* DOOR02 - Porta secondaria *)*)
	fKEY_QE_ST		:FLT_TAP; (* DOOR03 - Quadro Elettrico *)

END_VAR
(*************** ISPESL *****************)
(*
fALARM_PB(IN:=ALARM_PB);
IF fALARM_PB.EVH THEN
	LogEv(EL_AlarmStop,EO_PBV,1,1,'Over_Pressure_Alarm');
END_IF

fALARM_TB(IN:=ALARM_TB);
IF fALARM_TB.EVH THEN
	LogEv(EL_AlarmStop,EO_TBV,1,1,'Over_Temperature_Alarm');
END_IF

fALARM_PM(IN:=ALARM_PM);
IF fALARM_PM.EVH THEN
	LogEv(EL_AlarmStop,EO_PMV,1,1,'Under_Pressure_Alarm');
END_IF
*)
(****************************************)

(*### VPN Connection Check ###*)(*
fVPN_OUT1(IN:=VPN_OUT1);
IF fVPN_OUT1.EVH THEN
	LogEv(EL_Log,EO_VPN,1,1,'CONNECT_ON');
END_IF
IF fVPN_OUT1.EVL THEN
	LogEv(EL_Log,EO_VPN,1,2,'CONNECT_OFF');
END_IF*)

(*### VPN Status Check ###*)
fVPN_OUT2(IN:=VPN_OUT2);
IF fVPN_OUT2.EVH THEN
	LogEv(EL_Log,EO_VPN,1,3,'STATUS_UP');
END_IF
IF fVPN_OUT2.EVL THEN
	LogEv(EL_Wrn,EO_VPN,1,4,'STATUS_DOWN');
END_IF

(*### DOOR01 Status Check ###*)(*
fKEY_CT_ST(IN:=KEY_CT_ST);
IF fKEY_CT_ST.EVH THEN
	LogEv(EL_Log,EO_DOOR,1,2,'Centrale_termica_Close');
END_IF
IF fKEY_CT_ST.EVL THEN
	LogEv(EL_Wrn,EO_DOOR,1,1,'Centrale_termica_Open');
END_IF*)

(*### DOOR02 Status Check ###*)(*
fKEY_SCT_ST(IN:=KEY_SCT_ST);
IF fKEY_SCT_ST.EVH THEN
	LogEv(EL_Log,EO_DOOR,2,2,'Sottocentrale_termica_Close');
END_IF
IF fKEY_SCT_ST.EVL THEN
	LogEv(EL_Wrn,EO_DOOR,2,1,'Sottocentrale_termica_Open');
END_IF*)

(*### DOOR03 Status Check ###*)
fKEY_QE_ST(IN:=KEY_QE_ST);
IF fKEY_QE_ST.EVH THEN
	LogEv(EL_Log,EO_DOOR,3,2,'Quadro_Close');
END_IF
IF fKEY_QE_ST.EVL THEN
	LogEv(EL_Wrn,EO_DOOR,3,1,'Quadro_Open');
END_IF
END_PROGRAM

(* POU Utils Functions/FLT_TAP, ST *)
FUNCTION_BLOCK FLT_TAP
VAR_INPUT
	IN		: BOOL;
	TAP		: BYTE:=4;
	INITEV	: BOOL:=TRUE;
END_VAR
VAR_OUTPUT
	OUT		: BOOL;
	EVH		: BOOL;
	EVL		: BOOL;
END_VAR
VAR
	init	: BOOL:=FALSE;
	cnt		: BYTE;
END_VAR
EVH:=FALSE;
EVL:=FALSE;

IF NOT init THEN
	init := TRUE;
	IF INITEV THEN
		OUT  := NOT IN;
		cnt  := TAP;
	ELSE
		OUT  := IN;
	END_IF
END_IF

IF OUT<>IN THEN
	cnt:=cnt+1;
	IF cnt>TAP THEN
		OUT:=IN;
		cnt:=0;
		IF OUT THEN EVH:=TRUE; ELSE EVL:=TRUE; END_IF
	END_IF
ELSE
	cnt:=0;
END_IF
END_FUNCTION_BLOCK

(* POU Utils Functions/AVERAGE_T, ST *)
FUNCTION_BLOCK AVERAGE_T
VAR_INPUT
	IN: 	INT;
END_VAR
VAR_OUTPUT
	HI:		INT;
	AVG:	INT;
	LOW:	INT;
	ERR:	BOOL;
END_VAR
VAR
	sum:	DINT;
	cnt:	WORD;
END_VAR
IF cnt>=65000 THEN
	ERR:=TRUE;
	Read();
	sum := sum - AVG;
	cnt := cnt + 1;
END_IF

sum := sum + IN;
cnt := cnt + 1;

IF IN<LOW THEN  LOW:=IN; END_IF
IF IN>HI  THEN HI :=IN; END_IF
END_FUNCTION_BLOCK
ACTION Read:
AVG := DINT_TO_INT(sum/cnt);
END_ACTION
ACTION Reset:
HI:=IN;
AVG:=IN;
LOW:=IN;
ERR:=FALSE;

sum:=IN;
cnt:=1;
END_ACTION

(* POU Utils Functions/COPY_32SWAP16, ST *)
FUNCTION COPY_32SWAP16:BOOL
VAR_INPUT
	pSourceAddress		:POINTER TO ARRAY[1..2] OF WORD;
	pDestinationAddress	:POINTER TO ARRAY[1..2] OF WORD;
END_VAR
VAR
END_VAR
pDestinationAddress^[1]:=pSourceAddress^[2];
pDestinationAddress^[2]:=pSourceAddress^[1];
END_FUNCTION

(* POU Utils Functions/FLT_EVENT, ST *)
FUNCTION_BLOCK FLT_EVENT
VAR_INPUT
	IN		: BOOL;
	INITEV	: BOOL:=TRUE;
END_VAR
VAR_OUTPUT
	EVH		: BOOL;
	EVL		: BOOL;
END_VAR
VAR
	init	: BOOL:=FALSE;
	old		: BOOL;
END_VAR
EVH:=FALSE;
EVL:=FALSE;

IF NOT init THEN
	init:=TRUE;
	IF INITEV THEN
		old := NOT IN;
	ELSE
		old := IN;
	END_IF
END_IF

IF old<>IN THEN
	old:=IN;
	IF IN THEN EVH:=TRUE; ELSE EVL:=TRUE; END_IF
END_IF
END_FUNCTION_BLOCK

(* POU Utils Functions/FLT_TIME, ST *)
FUNCTION_BLOCK FLT_TIME
VAR_INPUT
	IN		: BOOL;
	TTAP	: TIME:=T#5s;
	INITEV	: BOOL:=TRUE;
END_VAR
VAR_OUTPUT
	OUT		: BOOL;
	EVH		: BOOL;
	EVL		: BOOL;
END_VAR
VAR
	init	: BOOL:=FALSE;
	timer	: TON;
END_VAR
EVH:=FALSE;
EVL:=FALSE;

IF NOT init THEN
	init := TRUE;
	IF INITEV THEN
		OUT  := NOT IN;
	ELSE
		OUT  := IN;
	END_IF
END_IF

IF OUT<>IN THEN
	timer(IN:=TRUE,PT:=TTAP);
	IF timer.Q THEN
		OUT:=IN;
		timer(IN:=FALSE);
		IF OUT THEN EVH:=TRUE; ELSE EVL:=TRUE; END_IF
	END_IF
ELSE
	timer(IN:=FALSE);
END_IF
END_FUNCTION_BLOCK

(* POU TCP_Logger/LogTrig, ST *)
FUNCTION LogTrig : BOOL
VAR
	s1 : STRING(160);
	i  : BYTE;
	j  : WORD;
END_VAR
(*---------------------------------------------------------------*)
(*---------------------------------------------------------------*)
Logger.TLen:=0;
(* Set GET header *)
ADDSTRING(ADR(Logger.TData), ADR(Logger_GETSTART), Logger.TLen);

(* Insert Header *)
s1:=INSERT('ID=&V=1&D=',DWORD_TO_STRING(Plant_SN),3);
s1:=CONCAT(s1,Sys.Time_LogString);
s1:=CONCAT(s1,'&S=');
IF Sys.Alarm THEN i:=2; ELSIF Sys.Warning THEN i:=1; ELSE i:=0; END_IF
s1:=CONCAT(s1,BYTE_TO_STRING(i));
ADDSTRING(ADR(Logger.TData), ADR(s1), Logger.TLen);

(* Insert contabilizers  *)
GAS01.AddLogData( MODBUS:=MODB01 );
CTB01.AddLogData( MBUS:=MBUS01 );
CTB02.AddLogData( MBUS:=MBUS01 );
CTB03.AddLogData( MBUS:=MBUS01 );
CTB04.AddLogData( MBUS:=MBUS01 );

(* Finalize string *)
ADDSTRING(ADR(Logger.TData), ADR(Logger_GETEND), Logger.TLen);

(*---------------------------------------------------------------*)
(*---------------------------------------------------------------*)

Logger_Send();
END_FUNCTION

(* POU Utils Functions/MEMCLR, ST *)
FUNCTION MEMCLR:BOOL
VAR_INPUT
	pDestinationAddress:POINTER TO ARRAY[1..2] OF BYTE;
	BytesToClear:WORD;
END_VAR
VAR
END_VAR
WHILE (BytesToClear > 0) DO
	pDestinationAddress^[1]:=0;
	pDestinationAddress:=ADR(pDestinationAddress^[2]); (* increment destination *)
	BytesToClear:=BytesToClear -1; (* decrement number of bytes to copy *)
END_WHILE
END_FUNCTION

(* POU Plant_Objects/obj_CAL_ROBUR_AY, ST *)
FUNCTION_BLOCK obj_CAL_ROBUR_AY (* CALDAIA ROBUR AY from DDC *)
VAR_INPUT
	(* Settings *)
	ID				: BYTE; (* Index of instanced object *)
	NetID			: WORD; (* Network ID on ROBUR DDC *)

	(* Controls *)
	Rearm			: BOOL; (* 40244=UID(u16-Unit), 40245=1(u16-Reset) *)

	(* States *)
	OnOff			: WORD; (* 12028 + 0*64 *)
	TSend			: INT;	(* 35023 + 0*250 *)
	TRet			: INT;	(* 35024 + 0*250 *)
	Power			: WORD; (* 35044 + 0*250 = Power feedback percentage 0-100% *)
	Status			: WORD; (* 35061 + 0*250 = General alarm bits1&0 00:OK 01:LOG 10:WRN 11:ERR *)

END_VAR
VAR_OUTPUT
	(* Visu/Log *)
	Status_Log		: BYTE;
	Status_Vis : DWORD;
END_VAR
VAR
END_VAR
(* Status color *)
   IF (Status AND 16#3)=16#3 THEN Status_Log:=2; Status_Vis:=16#2020F0;
ELSIF (Status AND 16#3)>1    THEN Status_Log:=1; Status_Vis:=16#20F0F0;
              				 ELSE Status_Log:=0; Status_Vis:=SEL(OnOff=1,16#006000,16#20F020);
END_IF
END_FUNCTION_BLOCK

(* POU Plant_Objects/obj_CIR, ST *)
FUNCTION_BLOCK obj_CIR
VAR_INPUT
	(* Settings *)
	ID				: BYTE;
	Chk_CntTrig		: BYTE:=10;	(* Check error trigger 5s *)
	(* Controls *)
	Ctrl_SetPoint 	: INT;
(*	CIR_RUN			: BOOL; (* Standard run request *) *)
	CIR_RUN_REQ		: BOOL; (* External run request (no heat or cold requested) *)
	CIR_STOP_REQ	: BOOL; (* External stop request (has priority over RUN signals!) *)
	(* Physical inputs *)
	CIR_AL			: BOOL; (* Alarm input signal *)
	CIR_ST			: BOOL; (* Status input signal *)
	CIR_AUTO		: BOOL; (* Auto/Manual input signal *)
END_VAR
VAR_IN_OUT
END_VAR
VAR_OUTPUT
	(* Physical outputs *)
	CIR_EN			: BOOL;		(* CIR control output *)
	(* Status *)
	Run				: BOOL;		(* Running signal for CALs *)
	Status_Log		: BYTE;
	Status_Vis 		: DWORD;
END_VAR
VAR
	InitOK			: BOOL;
	Ctrl_Run		: BOOL;

	StartDelay		: BYTE; (* Start delay ID based to avoid peak overload *)
	StopDelay		: TOF;  (* Stop delay PLANT based for boiler heat at shutdown *)

	fCIR_AL			: FLT_TAP := ( TAP:=10, INITEV:=FALSE );
	fCIR_ST_ERR		: FLT_TAP := ( TAP:=10, INITEV:=FALSE );
	fCIR_AUTO		: FLT_TAP := ( TAP:= 5, INITEV:=FALSE );
END_VAR
(* Check initialization *)
IF NOT InitOK THEN Init(); END_IF

(* Set running flag *)
IF T_AMB<Plant_MaxRunTAmb THEN
	(* Open Control Loop [TEMPORARY] *)
	IF Ctrl_SetPoint<180 THEN Ctrl_Run:=FALSE; StartDelay:=ID;
	ELSE
		IF StartDelay>2 THEN
			Ctrl_Run:=FALSE;
			StartDelay:=StartDelay-2;
		ELSE
			Ctrl_Run:=TRUE;
		END_IF
	END_IF
	(* ==> Future obj_TERM (Thermostat) function will be an external object <== *)
ELSE
	Ctrl_Run:=FALSE;
	StartDelay:=ID;
END_IF

(* Antifreeze function: reload off delay *)
IF T_AMB<Plant_AntiFreezeTAmb THEN
	StopDelay(IN:=TRUE);
END_IF

(* Set delayed output *)
StopDelay(IN:=Ctrl_Run, PT:=Plant_CirOffDelay);
   IF CIR_STOP_REQ THEN CIR_EN:=FALSE;
ELSIF CIR_RUN_REQ  THEN CIR_EN:=TRUE;
				   ELSE CIR_EN:=StopDelay.Q; END_IF

(* Check errors *)
fCIR_AL(IN:=CIR_AL);
IF fCIR_AL.EVH THEN LogEv(EL_Alarm,EO_CAL,ID,3,'CIR_Alarm'); END_IF
IF fCIR_AL.EVL THEN LogEv(EL_Log  ,EO_CAL,ID,4,'CIR_Alarm_Recover'); END_IF

fCIR_ST_ERR(IN:=(CIR_ST<>CIR_EN));
IF fCIR_ST_ERR.EVH THEN
	IF CIR_AUTO THEN
		LogEv(SEL(CIR_ST,EL_Alarm,EL_Wrn),EO_CIR,ID,SEL(CIR_ST,5,6),'CIR_Status');
	ELSE
		LogEv(EL_Wrn,EO_CIR,ID,SEL(CIR_ST,1,2),'CIR_Manual_Wrn');
	END_IF
END_IF

fCIR_AUTO(IN:=CIR_AUTO);
IF fCIR_AUTO.EVL THEN LogEv(EL_Wrn,EO_CIR,ID,7,'CIR_Manual'); END_IF
IF fCIR_AUTO.EVH THEN LogEv(EL_Log,EO_CIR,ID,8,'CIR_Auto'  ); END_IF


(* Set RUN signal (for external objects) *)
IF fCIR_AL.OUT OR fCIR_ST_ERR.OUT THEN
	Run:=FALSE;
ELSE
	Run:=Ctrl_Run;
END_IF


(* Status color *)
   IF fCIR_AL.OUT			 				 THEN Status_Log:=2; Status_Vis:=16#2020F0;
ELSIF fCIR_ST_ERR.OUT OR fCIR_AUTO.OUT=FALSE THEN Status_Log:=1; Status_Vis:=16#20F0F0;
                  	   				 		 ELSE Status_Log:=0; Status_Vis:=SEL(CIR_EN,16#006000,16#20F020);
END_IF
END_FUNCTION_BLOCK
ACTION Init:
(* End initialization *)
InitOK:=TRUE;
END_ACTION

(* POU Plant_Objects/obj_CRON, ST *)
FUNCTION_BLOCK obj_CRON (* CRONO-TERMOSTATO *)
VAR_INPUT
	(* Settings *)
	ID			: BYTE;		(* Index of instanced object *)

	InitOK		: BOOL;
	Alarm		: BOOL;
	Warning		: BOOL;

	Profile		: typ_Cron_Profile; 				(* Profilo attivo *)
	ProfileNr	: BYTE;								(* Indice profilo attivo *)
	CalendarIdx : WORD;								(* Indice calendario attivo *)
	Jolly		: ARRAY[0..9] OF typ_Cron_Jolly;	(* Jolly attivi *)

END_VAR
VAR_IN_OUT
END_VAR
VAR_OUTPUT
	SetPoint		: INT;
	(* Status *)
	Status_Log		: BYTE;
	Status_Vis 		: DWORD;
END_VAR
VAR
	Buf: 	ARRAY[0..512] OF BYTE;
	hFile: 	DWORD;
	sFile: 	STRING;
	sFile2: STRING;

	i:		WORD;
	t1:		DWORD;
	t2:		BOOL;

END_VAR
(* Check initialization *)
IF NOT InitOK THEN Init(); END_IF

(* Chrono *)
IF CalendarIdx<>Sys.Time_CT_Day THEN DB_Load(); END_IF
SetPoint:=Profile.Setpoint[Sys.Time_CT_Quarter];

(* Check jolly *)
FOR i := 0 TO 9 DO
	IF ( DT_TO_DWORD(Jolly[i].Start)>0  AND Jolly[i].End>Jolly[i].Start AND
	     Jolly[i].Start<=Sys.Time_CT_DT AND Jolly[i].End>Sys.Time_CT_DT ) THEN
			SetPoint:=Jolly[i].Temp;
	END_IF
END_FOR


(* Status color *)
   IF Alarm   THEN Status_Log:=2; Status_Vis:=16#2020F0;
ELSIF Warning THEN Status_Log:=1; Status_Vis:=16#20F0F0;
              ELSE Status_Log:=0; Status_Vis:=16#20F020;
			  END_IF
END_FUNCTION_BLOCK
ACTION DB_Create:
(* Check presence of previous year *)
sFile2:=REPLACE(STR1:=sFile, STR2:=WORD_TO_STRING(Sys.Time_Year-1), L:=4, P:=LEN(FilesPath)+1);
hFile:=SysFileOpen(FileName:=sFile2, Mode:='r');
IF hFile<>0 THEN
	(* Check file version and close *)
	SysFileRead(File:=hFile, Buffer:=ADR(Buf), Size:=1);
	SysFileClose(File:=hFile);
END_IF
IF hFile<>0 AND Buf[0]=1 THEN
	(* Copy file *)
	SysFileCopy(FileDest:=sFile, FileSource:=sFile2);
ELSE
	(* Create empty file *)
	hFile:=SysFileOpen(FileName:=sFile, Mode:='w');
	MEMCLR(pDestinationAddress:=ADR(Buf), BytesToClear:=SIZEOF(Buf));
	FOR i := 0 TO 10239 BY 512 DO
		t1:=SysFileWrite(File:=hFile, Buffer:=ADR(Buf), Size:=512);
	END_FOR
	Buf[0]:=1;
	t2:=SysFileSetPos(File:=hFile, Pos:=0);
	t1:=SysFileWrite(File:=hFile, Buffer:=ADR(Buf), Size:=1);
	SysFileClose(File:=hFile);
END_IF
END_ACTION
ACTION DB_Load:
DB_SetName();

(* Open data file *)
hFile:=SysFileOpen(FileName:=sFile, Mode:='r');

(* File not found *)
IF hFile=0 THEN
	Warning:=TRUE;
	LogEv(EL_Wrn,EO_CRON,ID,1,'No_data_file');
	DB_Create();
	(* Reopen file *)
	hFile:=SysFileOpen(FileName:=sFile, Mode:='r');
	IF hfile=0 THEN
		Alarm:=TRUE;
		LogEv(EL_Alarm,EO_CRON,ID,3,'Filesystem_error');
		RETURN;
	END_IF
END_IF

(* Check version *)
SysFileRead(File:=hFile, Buffer:=ADR(Buf), Size:=1);
IF Buf[0]<>1 THEN
	IF NOT Alarm THEN
		Alarm:=TRUE;
		LogEv(EL_Alarm,EO_CRON,ID,2,'Bad_data_version');
	END_IF
	SysFileClose(File:=hFile);
	RETURN;
END_IF

(* Read Jolly data *)
t2:=SysFileSetPos(File:=hFile, Pos:=512);
t1:=SysFileRead(File:=hFile, Buffer:=ADR(Jolly), Size:=SIZEOF(Jolly));
(* Read active profile index *)
CalendarIdx:=Sys.Time_CT_Day;
t2:=SysFileSetPos(File:=hFile, Pos:=(1024+4*CalendarIdx));
t1:=SysFileRead(File:=hFile, Buffer:=ADR(ProfileNr), Size:=SIZEOF(ProfileNr));
(* Read active profile *)
t2:=SysFileSetPos(File:=hFile, Pos:=(3072+512*ProfileNr));
t1:=SysFileRead(File:=hFile, Buffer:=ADR(Profile), Size:=SIZEOF(Profile));

(* Close file and validate data *)
SysFileClose(File:=hFile);
END_ACTION
ACTION DB_SetName:
(* Create current filename 'yyyyCRnn.DAT' *)
sFile:=CONCAT(FilesPath,WORD_TO_STRING(Sys.Time_Year));
sFile:=CONCAT(STR1:=sFile, STR2:='CR');
IF ID<10 THEN
sFile:=CONCAT(STR1:=sFile, STR2:='0');
END_IF
sFile:=CONCAT(STR1:=sFile, STR2:=BYTE_TO_STRING(ID));
sFile:=CONCAT(STR1:=sFile, STR2:='.DAT');
END_ACTION
ACTION Init:
DB_Load();
InitOK:=TRUE;
END_ACTION

(* POU Plant_Objects/obj_CRON_EDITOR, ST *)
FUNCTION_BLOCK obj_CRON_EDITOR
VAR_INPUT

	(* Common selections *)
	CN_Sel:			BYTE:=1;
	CN_Act:			BYTE;
	CN_YSel:		WORD:=2015;
	CN_YAct:		WORD;

	(* Profile editor *)
	PR_Sel: 		BYTE:=1;
	PR_Act:			BYTE;
	PR_TT:			REAL;
	PR:				typ_Cron_Profile;
	(* Profile signals *)
	PR_Load:		BOOL;
	PR_Save:		BOOL;

	(* Calendar editor *)
	CA_Sel:			BYTE:=1; (* Calendar month selected *)
	CA_Act:			BYTE;    (* Calendar month active *)
	CA_DayF:		BYTE:=0;
	CA_DayL:		BYTE:=31;
	CA_TPR:			BYTE;
	CA:				typ_Cron_Calendar; (* Only used for first 32 entries *)
	(* Calendar signals *)
	CA_Load:		BOOL;
	CA_Save:		BOOL;

	(* Jolly editor *)
	JL:				ARRAY[0..9] OF typ_Cron_Jolly;
	(* Jolly signals *)
	JL_Load:		BOOL;
	JL_Save:		BOOL;

END_VAR
VAR_OUTPUT
	Message		: STRING;
END_VAR
VAR
	sFileName	: STRING;
	sFileMode	: STRING;
	hFile		: DWORD;

	i			: WORD;
	ver			: BYTE;
	r1			: BOOL;
	r2			: DWORD;

END_VAR
IF PR_Load THEN PR_Load_Exe(); PR_Load:=FALSE; END_IF
IF PR_Save THEN PR_Save_Exe(); PR_Save:=FALSE; END_IF
IF CA_Load THEN CA_Load_Exe(); CA_Load:=FALSE; END_IF
IF CA_Save THEN CA_Save_Exe(); CA_Save:=FALSE; END_IF
IF JL_Load THEN JL_Load_Exe(); JL_Load:=FALSE; END_IF
IF JL_Save THEN JL_Save_Exe(); JL_Save:=FALSE; END_IF
END_FUNCTION_BLOCK
ACTION CA_Load_Exe:
sFileMode:='r';
FileOpen();

IF hFile<>0 THEN

	(* Read calendar month *)
	FOR i := 0 TO 31 DO
		r1:=SysFileSetPos(File:=hFile, Pos:=(1024 + ((CA_Sel-1)*32 + i)*4));
		r2:=SysFileRead(File:=hFile, Buffer:=ADR(CA.Profile[i]), Size:=1);
	END_FOR

	(* Close file *)
	SysFileClose(File:=hFile);

	(* Validate data *)
	CA_Act :=CA_Sel;
	CN_Act :=CN_Sel;
	CN_YAct:=CN_YSel;

	Message:='Calendar load OK';

END_IF
END_ACTION
ACTION CA_Save_Exe:
sFileMode:='a';
FileOpen();

IF hFile<>0 THEN

	(* Write calendar month *)
	FOR i := 0 TO 31 DO
		r1:=SysFileSetPos(File:=hFile, Pos:=(1024 + ((CA_Sel-1)*32 + i)*4));
		r2:=SysFileGetPos(hFile);
		r2:=SysFileWrite(File:=hFile, Buffer:=ADR(CA.Profile[i]), Size:=1);
	END_FOR

	(* Close file *)
	SysFileClose(File:=hFile);

	Message:='Calendar save OK';

END_IF
END_ACTION
ACTION FileOpen:
(* Create current filename 'yyyyCRnn.DAT' *)
sFileName:=CONCAT(FilesPath,WORD_TO_STRING(CN_YSel));
sFileName:=CONCAT(STR1:=sFileName, STR2:='CR');
IF CN_Sel<10 THEN
sFileName:=CONCAT(STR1:=sFileName, STR2:='0');
END_IF
sFileName:=CONCAT(STR1:=sFileName, STR2:=BYTE_TO_STRING(CN_Sel));
sFileName:=CONCAT(STR1:=sFileName, STR2:='.DAT');

(* Check file version and size! *)
(* ... *)

(* Open data file *)
hFile:=SysFileOpen(FileName:=sFileName, Mode:='r');

(* File not found *)
IF hFile=0 THEN
	Message:='File not found';
	RETURN;
END_IF

(* Close file *)
SysFileClose(File:=hFile);

(* Open data file *)
hFile:=SysFileOpen(FileName:=sFileName, Mode:=sFileMode);
END_ACTION
ACTION JL_Load_Exe:
sFileMode:='r';
FileOpen();

IF hFile<>0 THEN

	(* Read jolly *)
	r1:=SysFileSetPos(File:=hFile, Pos:=512);
	r2:=SysFileRead(File:=hFile, Buffer:=ADR(JL), Size:=SIZEOF(JL));

	(* Close file *)
	SysFileClose(File:=hFile);

	(* Validate data *)
	CN_Act:=CN_Sel;
	CN_YAct:=CN_YSel;

	Message:='Jolly load OK';

END_IF
END_ACTION
ACTION JL_Save_Exe:
sFileMode:='a';
FileOpen();

IF hFile<>0 THEN

	(* Write selected profile *)
	r1:=SysFileSetPos(File:=hFile, Pos:=512);
	r2:=SysFileWrite(File:=hFile, Buffer:=ADR(JL), Size:=SIZEOF(JL));

	(* Close file *)
	SysFileClose(File:=hFile);

	Message:='Jolly save OK';

END_IF
END_ACTION
ACTION PR_Load_Exe:
sFileMode:='r';
FileOpen();

IF hFile<>0 THEN

	(* Read selected profile *)
	r1:=SysFileSetPos(File:=hFile, Pos:=(3072 + 512*PR_Sel));
	r2:=SysFileRead(File:=hFile, Buffer:=ADR(PR), Size:=SIZEOF(PR));

	(* Close file *)
	SysFileClose(File:=hFile);

	(* Validate data *)
	PR_Act:=PR_Sel;
	CN_Act:=CN_Sel;
	CN_YAct:=CN_YSel;

	Message:='Profile load OK';

END_IF
END_ACTION
ACTION PR_Save_Exe:
sFileMode:='a';
FileOpen();

IF hFile<>0 THEN

	(* Write selected profile *)
	r1:=SysFileSetPos(File:=hFile, Pos:=(3072 + 512*PR_Sel));
	r2:=SysFileWrite(File:=hFile, Buffer:=ADR(PR), Size:=SIZEOF(PR));

	(* Close file *)
	SysFileClose(File:=hFile);

	Message:='Profile save OK';

END_IF
END_ACTION

(* POU Plant_Objects/obj_CTL, ST *)
FUNCTION_BLOCK obj_CTL
VAR_INPUT
	(* Settings *)
	ID				: BYTE;	(* Index of instanced object *)
	(* Physical inputs *)
	CTL_ST			: BOOL;
END_VAR
VAR_IN_OUT
	COUNT			: DWORD;
END_VAR
VAR_OUTPUT
	(* Status *)
	Status_Log		: BYTE;
END_VAR
VAR
	Filter			: FLT_TAP := ( INITEV:=FALSE );
	Timer			: TON;
	TCount			: DWORD;
	i				: DWORD;
END_VAR
(* Execute timer *)
Timer(IN:=NOT Timer.Q, PT:=T#60m);
(* Execute filter *)
Filter(IN:=CTL_ST);
(* Count event *)
IF Filter.EVH THEN
	COUNT:=COUNT+1;
	TCount:=TCount+1;
	(* Check flow rate *)
	IF TCount>=Plant_MaxWaterLoss THEN
		i:=(TCount*TIME_TO_DWORD(Timer.PT))/TIME_TO_DWORD(Timer.ET);
		LogEv(EL_AlarmStop,EO_CTL,ID,1,DWORD_TO_STRING(i));
		Status_Log:=2;
		TCount:=0;
		Timer(IN:=FALSE);
	END_IF
END_IF
(* Check timer *)
IF Timer.Q THEN
	TCount:=0;
	IF TCount<Plant_MaxWaterLoss THEN
		Status_Log:=0;
	END_IF
END_IF
END_FUNCTION_BLOCK

(* POU Plant_Objects/obj_GAS, ST *)
FUNCTION_BLOCK obj_GAS

VAR_INPUT
	(* Settings *)
	ID				: BYTE;
	DI_Input		: BOOL;	(* Ingresso Digitale per il conteggio  *)
	Peso			: INT;	(* Peso dell' impulso , serve per avere una lettura immediata dell'unità ingegneristica *)
	TempoTimeOut	: TIME;	(* Minuti di inattività per la segnalazione del WRN *)
END_VAR
VAR_OUTPUT
	WRN				: BOOL;	(* Segnalazione Warning *)
	(* Status *)
	Status_Log		: BYTE;
	Status_Vis 		: DWORD;
END_VAR
VAR
	TRig_DI			: R_TRIG;
	TimeOut			: TON;
	TRigR_TimeOut	: R_TRIG;
	TRigL_TimeOut	: F_TRIG;
END_VAR
VAR_IN_OUT
                Contatore                          : DINT;
                Totalizzatore    			 :DINT; (* Totale Conteggio x valore peso *)
END_VAR
(* MANCA UN MINIMO DI TAP ==> meglio usare FLT_TAP per detect fronte di salita *)

(* Triggero sul fronte di salita l'ingresso digitale *)
TRig_DI(CLK:=DI_Input );

(* Conto i fronti di salita  in modo de creare rapporto*)
IF  TRig_DI.Q THEN
	Contatore:=Contatore+1;
	Totalizzatore:=Contatore*Peso;
END_IF

(* Imposto il time out se non c'è movimento sulla linea per il tempo impostato loggo un Warning *)
TimeOut(IN:=NOT DI_Input , PT:=TempoTimeOut, Q=> , ET=> );
TRigR_TimeOut( CLK:= TimeOut.Q  );
TRigL_TimeOut( CLK:= TimeOut.Q  );

		IF  TRigR_TimeOut.Q THEN     (* Condizione di WARNING *)
					WRN:=TRUE;
 					LogEv(EL_Wrn,EO_GAS,ID,2,'Nessun_Movimento');
		END_IF

		IF  TRigL_TimeOut.Q THEN     (* Condizione di Rientro dal WARNING *)
					WRN:=FALSE;
 					LogEv(EL_Log,EO_GAS,ID,1,'');
		END_IF
END_FUNCTION_BLOCK

(* POU Plant_Objects/obj_MBUS, ST *)
FUNCTION_BLOCK obj_MBUS
(* === M-BUS PROTOCOL INTERFACE ===
   v1.0[16/03/05] - Added interface errors
*)
VAR_INPUT
	(* Settings *)
	ID				: BYTE;
	COM				: BYTE;
	BAUDRATE		: COM_BAUDRATE;
	(* Interface *)
	MBus 			: typMBus;
	MBus_Master 	: FbMBusMaster;
END_VAR
VAR_OUTPUT
	(* Status *)
	Status_Log		: BYTE;
	Status_Vis 		: DWORD;
END_VAR
VAR
	Alarm			: FLT_EVENT;
END_VAR
MBus_Master( bCOMPORT:=COM , enumBAUDRATE:=BAUDRATE , utMBus:=MBus );

(* Check status *)
Alarm(IN:=(MBus.bCOM_ERROR<>0));
IF Alarm.EVH THEN
	LogEv(EL_Alarm,EO_MBUS,ID,1,BYTE_TO_STRING(MBus.bCOM_ERROR));
END_IF
IF Alarm.EVL THEN
	LogEv(EL_Log,EO_MBUS,ID,2,'MBUS_OK');
END_IF

(* Log/visu status *)
   IF Alarm.IN   					THEN Status_Log:=2; Status_Vis:=16#2020F0;
ELSIF (MBus.bL1_ERROR AND 16#1F)<>0 THEN Status_Log:=1; Status_Vis:=16#20F0F0;
  				 					ELSE Status_Log:=0; Status_Vis:=16#20F020;
END_IF
END_FUNCTION_BLOCK

(* POU Plant_Objects/obj_MBUS_CTB_SCANNER, ST *)
FUNCTION_BLOCK obj_MBUS_CTB_SCANNER
VAR_INPUT
	(* Settings *)
	ID				: BYTE;
	EndScanAddress	: BYTE:=250;
	EndlessRescan   : BOOL:=FALSE;
	ScanPause		: TIME:=t#500ms;
	(* Controls *)
	Refresh			: BOOL; (* Enable automatic refresh of detected CTBs *)
	Rescan			: BOOL; (* Perform complete search for list-update *)
END_VAR
VAR_IN_OUT
	MBUS			: obj_MBUS;
END_VAR
VAR_OUTPUT
	ConnectedCTBs	: BYTE; (* Number of connected CTBs at last rescan *)
	(* Status *)
	Status_Log		: BYTE;
	Status_Vis 		: DWORD;
END_VAR
VAR

	(* Virtual contabilizer for scanner *)
	M1			: FbMBus_Heat;
	M1_Start	: BOOL;

	(* Da definire come datatype *)
(*	CTBS	: ARRAY [0..255] OF typ_MBUS_CTBS; *)
	NodoMBusPresente		: ARRAY [0..255] OF BOOL;
	ErroreNodoMBus			: ARRAY [0..255] OF BYTE;
	Status_Log_NodoMBus		: ARRAY [0..255] OF BYTE;
	Status_Vis_NodoMBus		: ARRAY [0..255] OF DWORD;
	CTB_utMBInfo			: ARRAY [0..255] OF typMBusInfo;
	CTB_utFTemp	 			: ARRAY [0..255] OF typMBusRecord;
	CTB_utRTemp	 			: ARRAY [0..255] OF typMBusRecord;
	CTB_utPower	 			: ARRAY [0..255] OF typMBusRecord;
	CTB_utFlow	 			: ARRAY [0..255] OF typMBusRecord;
	CTB_utEnergy 			: ARRAY [0..255] OF typMBusRecord;
	CTB_utVolume 			: ARRAY [0..255] OF typMBusRecord;
	CTB_utDTemp	 			: ARRAY [0..255] OF typMBusRecord;
	VisuDatiMbus			: ARRAY [0..255] OF typ_VisuStrutturaMbus;

	sta		 : BYTE; 	(* Status: 0:Idle, 1:Wait scan response, 2:Wait refresh response, 3:Wait refresh delay *)
	cnt		 : BYTE;	(* Selection counter *)
	pass_cnt : BYTE;	(* Active counter *)
	dly 	 : TON;
	s1 		 : STRING;
END_VAR
CASE sta OF
	0:
		IF NOT M1_Start THEN
			IF Rescan THEN
				(* Start scanning - with fast timeout and only one retry *)
				cnt:=0;
				pass_cnt:=0;
				MBUS.MBus_Master.bRetries:=1;
				MBUS.MBus_Master.tTimeout:=T#500ms;
				M1.dwAdr:=cnt;
				M1_Start:=TRUE;
				sta:=1;
			ELSIF Refresh THEN
				(* Start refresh *)
				cnt:=0;
				GoToNextActive();
				IF cnt>EndScanAddress THEN
					Refresh:=FALSE;
				ELSE
					MBUS.MBus_Master.bRetries:=3;
					MBUS.MBus_Master.tTimeout:=T#1000ms;
					M1.dwAdr:=cnt;
					M1_Start:=TRUE;
					sta:=2;
				END_IF
			END_IF
		END_IF

	1:
		IF NOT Rescan THEN
			sta:=0;
		ELSE
			IF NOT M1_Start THEN
				(* Get scan result *)
				UpdateNode();
				UpdateVisu();
				(* Next object *)
				cnt:=cnt+1;
				IF cnt>EndScanAddress THEN
					ConnectedCTBs:=pass_cnt;
					Rescan:=EndlessRescan;
					sta:=0;
				ELSE
					M1.dwAdr:=cnt;
					M1_Start:=TRUE;
				END_IF;
			END_IF
		END_IF

	2:
		IF NOT Refresh OR Rescan THEN
			sta:=0;
		ELSE
			IF NOT M1_Start THEN
				(* Get scan result *)
				UpdateNode();
				UpdateVisu();
				(* Next object *)
				cnt:=cnt+1;
				GoToNextActive();
				IF cnt>EndScanAddress THEN
					sta:=3;
					dly(IN:=FALSE, PT:=ScanPause);
				ELSE
					M1.dwAdr:=cnt;
					M1_Start:=TRUE;
				END_IF;
			END_IF
		END_IF

	3:
		(* Refresh cycle delay *)
		dly(IN:=TRUE, PT:=ScanPause);
		IF dly.Q THEN sta:=0; END_IF

ELSE
	sta:=0;
END_CASE

(* Update virtual contabilizer *)
M1( (*dwAdr:= cnt,*) xSND_NKE:=TRUE , utMBus:=MBUS.MBus , xStart:=M1_Start );
END_FUNCTION_BLOCK
ACTION GoToNextActive:
WHILE NodoMBusPresente[cnt] <> TRUE AND cnt<=EndScanAddress DO
	cnt:=cnt+1;
END_WHILE
END_ACTION
ACTION UpdateNode:
ErroreNodoMBus[cnt]:=M1.bError;
CTB_utMBInfo[cnt]:=M1.utMBInfo;
CTB_utEnergy[cnt]:=M1.utEnergy;
CTB_utPower [cnt]:=M1.utPower;
CTB_utVolume[cnt]:=M1.utVolume;
CTB_utFlow  [cnt]:=M1.utFlow;
CTB_utFTemp [cnt]:=M1.utFTemp;
CTB_utRTemp [cnt]:=M1.utRTemp;
CTB_utDTemp [cnt]:=M1.utDTemp;

				(* Check node status *)
				IF ErroreNodoMBus[cnt]<>0  THEN
           			(* se non sono in allarme di comunicazione loggo l'allarme *)
					IF Status_Log_NodoMBus[cnt]<>2 AND sta=2 THEN
						LogEv(EL_Alarm,EO_CTB,cnt,2,CONCAT('Err',BYTE_TO_STRING(ErroreNodoMBus[cnt])));
					END_IF
					(*se sono in fase di rescan memorizzo l'assenza del nodo *)
					IF sta=1 THEN NodoMBusPresente[cnt]:=FALSE;	END_IF
					(* Update status *)
					Status_Log_NodoMBus[cnt]:=2;
					Status_Vis_NodoMBus[cnt]:=16#2020F0;
		    	ELSE
					(* tutto OK Comunizaione andata a buon termine *)
					(* se non sono in allarme di comunicazione loggo l'allarme, ma  se non presente *)
					IF Status_Log_NodoMBus[cnt]<>0 AND sta=2 THEN
						LogEv(EL_Log,EO_CTB,cnt,1,'Nodo_OK');
					END_IF
					(*se sono in fase di rescan memorizzo la presenza del nodo *)
					IF sta=1 THEN NodoMBusPresente[cnt]:=TRUE; pass_cnt:=pass_cnt+1; END_IF
					(* Update status *)
					Status_Log_NodoMBus[cnt]:=0;
					Status_Vis_NodoMBus[cnt]:=16#20F020;
				END_IF
END_ACTION
ACTION UpdateVisu:
VisuDatiMbus[cnt].sdNodoPresente	:=SEL(NodoMBusPresente[cnt],'FAIL!','OK');
VisuDatiMbus[cnt].sdEnergia			:=CTB_utMBInfo[cnt].stMAN;
VisuDatiMbus[cnt].sdPotenza			:=CTB_utMBInfo[cnt].stMED;
VisuDatiMbus[cnt].sdVolume			:=CTB_utMBInfo[cnt].stID;

(*
VisuDatiMbus[cnt].sdEnergia			:=CONCAT(CTB_utEnergy[cnt].Value,CTB_utEnergy[cnt].Unit);
VisuDatiMbus[cnt].sdPotenza			:=CONCAT(CTB_utPower [cnt].Value,CTB_utPower [cnt].Unit);
VisuDatiMbus[cnt].sdVolume			:=CONCAT(CTB_utVolume[cnt].Value,CTB_utVolume[cnt].Unit);
VisuDatiMbus[cnt].sdFlow			:=CONCAT(CTB_utFlow  [cnt].Value,CTB_utFlow  [cnt].Unit);
VisuDatiMbus[cnt].sdTempIngresso	:=CONCAT(CTB_utFTemp [cnt].Value,CTB_utFTemp [cnt].Unit);
VisuDatiMbus[cnt].sdTempaUscita		:=CONCAT(CTB_utRTemp [cnt].Value,CTB_utRTemp [cnt].Unit);
VisuDatiMbus[cnt].sdTempDelta		:=CONCAT(CTB_utDTemp [cnt].Value,CTB_utDTemp [cnt].Unit);
*)

IF sta=1 AND NodoMBusPresente[cnt] THEN
(*	s1:=SEL(NodoMBusPresente[cnt],'FAIL','OK');*)
	s1:='FOUND';
	s1:=CONCAT(s1,'_');
	s1:=CONCAT(s1,CTB_utMBInfo[cnt].stMED);
	s1:=CONCAT(s1,'_');
	s1:=CONCAT(s1,CTB_utMBInfo[cnt].stID);
	LogEv(EL_Log,EO_CTB,cnt,100,s1);
END_IF
END_ACTION

(* POU Plant_Objects/obj_MBUS_CTB_SHARKY775, ST *)
FUNCTION_BLOCK obj_MBUS_CTB_SHARKY775
(* === M-BUS CONTABILIZER SHARKY 775 ===
   v1.0[16/03/05] - Error management
*)
VAR_INPUT
	(* Settings *)
	ID				: BYTE;
	ADDRESS			: DWORD;
	Refresh_Period	: TIME:=t#3m;
	(* Controls *)
	Refresh_Auto	: BOOL:=TRUE; (* Enable automatic refresh *)
	Refresh_Now		: BOOL; 	  (* Force an immediate refresh *)
END_VAR
VAR_IN_OUT
	(* Interface *)
	MBUS			: obj_MBUS;
END_VAR
VAR_OUTPUT
	M1				: FbMBus_Heat;
	(* Status *)
	Status_Log		: BYTE;
	Status_Vis 		: DWORD;
END_VAR
VAR
	dly 	 	: TON := (PT:=t#5s);
	M1_Start	: BOOL;

	init_st		: BOOL;
	bus_st0		: BYTE;
	dev_st0		: BYTE;

(*	S1			: FbMBusSend;
	S1_Start	: BOOL;*)
(*	C1			: FbUnitConverter; *)
END_VAR
(* Auto refresh timer *)
dly(IN:=NOT (dly.Q OR Refresh_Now OR (NOT Refresh_Auto)));
(* Trigger refresh *)
IF dly.Q OR Refresh_Now THEN
	dly.PT:=Refresh_Period;
	Refresh_Now:=FALSE;
	(* Start reading *)
	M1.dwAdr:= ADDRESS;
	M1.xSND_NKE:=TRUE;
	M1_Start:=TRUE;
END_IF

(* Contabilizer module *)
M1(	utMBus:=MBUS.MBus, xStart:=M1_Start );

(* Extra actions *)
(*C1( utMBus:=MBUS.MBus, xStart:=C1_Start );*)

(* Check status *)
IF NOT init_st OR M1.bError<>bus_st0 OR M1.utMBInfo.bMStatus<>dev_st0 THEN
	init_st:=TRUE;
	bus_st0:=M1.bError; dev_st0:=M1.utMBInfo.bMStatus;
	IF bus_st0<>0 THEN
		LogEv(EL_Alarm,EO_CTB,ID,2,BYTE_TO_STRING(bus_st0));
		Status_Log:=2; Status_Vis:=16#2020F0;
	ELSE
		IF dev_st0<>0 THEN
			Status_Log:=2; Status_Vis:=16#2020F0;
			CASE dev_st0 OF
				16#08: LogEv(EL_Alarm,EO_CTB,ID,10,'C-1');
				16#04: LogEv(EL_Alarm,EO_CTB,ID,10,'E-8');
				16#28: LogEv(EL_Alarm,EO_CTB,ID,10,'E-4');
				16#50: LogEv(EL_Alarm,EO_CTB,ID,10,'E-1');
				16#70: LogEv(EL_Alarm,EO_CTB,ID,10,'E-7');
				16#84: LogEv(EL_Alarm,EO_CTB,ID,10,'E-9');
				16#B0: LogEv(EL_Alarm,EO_CTB,ID,10,'E-3');
				16#D0: LogEv(EL_Alarm,EO_CTB,ID,10,'E-6');
				16#F0: LogEv(EL_Alarm,EO_CTB,ID,10,'Leak');
				16#10: LogEv(EL_Wrn  ,EO_CTB,ID,10,'E-5'); Status_Log:=1; Status_Vis:=16#20F0F0;
			ELSE
				LogEv(EL_Alarm,EO_CTB,ID,10,BYTE_TO_STRING(dev_st0));
			END_CASE
		ELSE
			Status_Log:=0; Status_Vis:=16#20F020;
			LogEv(EL_Log,EO_CTB,ID,1,'');
		END_IF
	END_IF
END_IF
END_FUNCTION_BLOCK
ACTION AddLogData:
Logger.s1:=INSERT('&CTB=',BYTE_TO_STRING(ID),4);
IF ID<10 THEN Logger.s1:=INSERT(Logger.s1,'0',4); END_IF

Logger.s1:=CONCAT(Logger.s1,M1.utFTemp.Value);		Logger.s1:=CONCAT(Logger.s1,';');
Logger.s1:=CONCAT(Logger.s1,M1.utRTemp.Value);		Logger.s1:=CONCAT(Logger.s1,';');
Logger.s1:=CONCAT(Logger.s1,M1.utFlow.Value);		Logger.s1:=CONCAT(Logger.s1,';');
Logger.s1:=CONCAT(Logger.s1,M1.utPower.Value);		Logger.s1:=CONCAT(Logger.s1,';');
Logger.s1:=CONCAT(Logger.s1,M1.utEnergy.Value);		Logger.s1:=CONCAT(Logger.s1,';');

Logger.s1:=CONCAT(Logger.s1,BYTE_TO_STRING(Status_Log));
ADDSTRING(ADR(Logger.TData), ADR(Logger.s1), Logger.TLen);
END_ACTION

(* POU Plant_Objects/obj_MODBUS, ST *)
FUNCTION_BLOCK obj_MODBUS
(* === MODBUS PROTOCOL INTERFACE ===
   v1.0[16/03/05] - Support for RS485 half-duplex
				  - Rewritten vars management with state machine
   v1.1[27/03/05] - Fixed vars manager & introduced retry before alarm
*)
VAR CONSTANT
	VARS_Max	: BYTE := 32;
END_VAR
VAR_INPUT
	(* Settings *)
	ID			: BYTE;
	COM			: BYTE;
	BAUDRATE	: COM_BAUDRATE;
	RS485		: BOOL := FALSE;
	(* Interface *)
	MB_MASTER	: MODBUS_EXTENDED_MASTER;
	MB_Start	: BOOL;
	MB_Query	: typModbusExtendedQuery;
	MB_Resp		: typModbusResponse;
	MB_Lock		: BOOL;
	(* Variables management *)
	VARS_En		: BOOL;
	VARS		: ARRAY [0..VARS_Max] OF typ_MODBUS_VAR;
	VARS_Check	: BOOL;
	VARS_Alarm	: BOOL;
END_VAR
VAR_OUTPUT
	(* Status *)
	Status_Log	: BYTE;
	Status_Vis	: DWORD;
END_VAR
VAR
	i			: BYTE;
	Alarm		: FLT_EVENT;
	VarTmr		: TON := (PT:=T#1s);
	VarSta		: BYTE; (* Status *)
	VarCnt		: BYTE; (* Scan counter *)
	VarRetry	: BYTE;
END_VAR
MB_MASTER(
	ENABLE:=TRUE ,
	ASCII_Mode:=FALSE,
	bCOM_PORT:=COM ,
	cbCOM_BAUDRATE:=BAUDRATE ,
	cpCOM_PARITY:=PARITY_NO ,
	csCOM_STOPBITS:=STOPBITS_1 ,
	cbsCOM_BYTESIZE:=BS_8 ,
	cfCOM_FLOW_CONTROL:=SEL(RS485,NO_FLOW_CONTROL,HALFDUPLEX) ,
	tTIME_OUT:=t#250ms ,
	StartFunction:=MB_Start ,
	ExtQuery:=MB_Query ,
	Response:=MB_Resp  );

(* Process variable management *)
IF VARS_En THEN VARS_Process(); END_IF

(* Check status *)
Alarm(IN:=(MB_MASTER.bInterfaceError<>0));
IF Alarm.EVH THEN
	LogEv(EL_Alarm,EO_MODBUS,ID,1,BYTE_TO_STRING(MB_MASTER.bInterfaceError));
END_IF
IF Alarm.EVL THEN
	LogEv(EL_Log,EO_MODBUS,ID,2,'MODBUS_OK');
END_IF

(* Log/visu status *)
   IF Alarm.IN   THEN Status_Log:=2; Status_Vis:=16#2020F0;
ELSIF Vars_Alarm THEN Status_Log:=1; Status_Vis:=16#20F0F0;
  				 ELSE Status_Log:=0; Status_Vis:=16#20F020;
END_IF
END_FUNCTION_BLOCK
ACTION VARS_Process:
(* Update var timers *)
VarTmr(IN:=(NOT VarTmr.Q));
IF VarTmr.Q THEN
	FOR i := 0 TO VARS_Max DO
		IF VARS[i].Refresh_Cnt>0 THEN VARS[i].Refresh_Cnt:=VARS[i].Refresh_Cnt-1; END_IF
	END_FOR
	VARS_Check:=TRUE;
END_IF


(* Process status *)
CASE VarSta OF
	0: (* === Init *)
		VarCnt:=0;
		VarSta:=1;

	1: (* === Wait check signal *)
		IF VARS_Check THEN
			VARS_Check:=FALSE;
			VarCnt:=0;
			VarSta:=2;
		END_IF

	2: (* === Check loop *)
		IF NOT (MB_Lock OR MB_Start) THEN
			WHILE VarCnt<=VARS_Max AND VarSta=2 DO
				(* Check only active vars *)
				IF VARS[VarCnt].SlaveAddress<>0 THEN
					(* Check var auto-refresh on timer checks *)
					IF VARS[VarCnt].Refresh_Time>0 AND VARS[VarCnt].Refresh_Cnt=0 THEN
						VARS[VarCnt].Refresh_Cnt:=VARS[VarCnt].Refresh_Time;
						VarSta:=3;
					END_IF
					(* Check refresh for change or request *)
					CASE VARS[VarCnt].FunCode OF
						16#5,16#6,16#F,16#10:
							IF VARS[VarCnt].Variable^<>VARS[VarCnt].Variable_Mirror THEN
								VARS[VarCnt].Variable_Mirror:=VARS[VarCnt].Variable^;
								VarSta:=3;
							END_IF
						16#1,16#2,16#3,16#4:
							IF VARS[VarCnt].Variable_Mirror<>0 THEN
								VARS[VarCnt].Variable_Mirror:=0;
								VarSta:=3;
							END_IF
					END_CASE
				END_IF
				(* Process query *)
				IF VarSta=3 THEN
					MB_Lock:=TRUE;
					MB_Query.SlaveAddress:=VARS[VarCnt].SlaveAddress;
					MB_Query.FunctionCode:=VARS[VarCnt].FunCode;
					CASE VARS[VarCnt].FunCode OF
						16#5,16#6,16#F,16#10:
							MB_Query.Read_StartAddress:=0;
							MB_Query.Read_Quantity:=0;
							MB_Query.Write_StartAddress:=VARS[VarCnt].FunAddress;
							MB_Query.Write_Quantity:=VARS[VarCnt].Variable_Size;
							MB_Query.Write_Data[0]:=VARS[VarCnt].Variable^;
						16#1,16#2,16#3,16#4:
							MB_Query.Read_StartAddress:=VARS[VarCnt].FunAddress;
							IF VARS[VarCnt].Variable_Size=200 THEN MB_Query.Read_Quantity:=2; ELSE
							  MB_Query.Read_Quantity:=VARS[VarCnt].Variable_Size;
							END_IF
							MB_Query.Write_StartAddress:=0;
							MB_Query.Write_Quantity:=0;
					END_CASE
					VarRetry:=0;
					MB_Start:=TRUE;
				ELSE
					VarCnt:=VarCnt+1;
				END_IF
			END_WHILE
			(* Check loop completed -> no actions *)
			IF VarSta=2 THEN VarSta:=1; END_IF
		END_IF

	3: (* === Wait & process MB response *)
		IF NOT MB_Start THEN
			IF MB_MASTER.MB_Error=0 THEN
				CASE VARS[VarCnt].FunCode OF
					16#1,16#2,16#3,16#4:
						IF VARS[VarCnt].Variable_Size=200 THEN
							COPY_32SWAP16(ADR(MB_Resp.Data), VARS[VarCnt].Variable);
						ELSIF VARS[VarCnt].Variable_Size>1 THEN
							MEMCPY(ADR(MB_Resp.Data), VARS[VarCnt].Variable, 2*VARS[VarCnt].Variable_Size);
						ELSE
							VARS[VarCnt].Variable^:=MB_Resp.Data[0];
						END_IF
				END_CASE
				MB_Lock:=FALSE;
				VarCnt:=VarCnt+1;
				VarSta:=2;
			ELSE
				IF VarRetry<3 THEN
					VarRetry:=VarRetry+1;
					MB_Start:=TRUE;
				ELSE
					IF VARS_Alarm=FALSE THEN
						LogEv(EL_Wrn,EO_MODBUS,ID,3,INT_TO_STRING(MB_MASTER.MB_Error));
						VARS_Alarm:=TRUE;
					END_IF
					MB_Lock:=FALSE;
					VarCnt:=VarCnt+1;
					VarSta:=2;
				END_IF
			END_IF
		END_IF

ELSE
	VarSta:=0;
END_CASE
END_ACTION

(* POU Plant_Objects/obj_MODBUS_ABB_DMTME72, ST *)
FUNCTION_BLOCK obj_MODBUS_ABB_DMTME72
VAR_INPUT
	(* Settings *)
	ID				: BYTE;
	ADDRESS			: BYTE:=31;
	Refresh_Period	: TIME:=t#3m;
	(* Controls *)
	Refresh_Auto	: BOOL:=TRUE; (* Enable automatic refresh *)
	Refresh_Now		: BOOL; 	  (* Force an immediate refresh *)
END_VAR
VAR_IN_OUT
	MODBUS			: obj_MODBUS;
END_VAR
VAR_OUTPUT
	Data			: typ_MODBUS_ABB_DMTME72;
	(* Status *)
	Status_Log		: BYTE;
	Status_Vis 		: DWORD;
END_VAR
VAR
	dly 	 : TON := (PT:=t#5s);
	sta		 : BYTE; 	(* Status *)



END_VAR
CASE sta OF
	0: (* === Wait update signals *)
		dly(IN:=NOT (dly.Q OR Refresh_Now OR (NOT Refresh_Auto)));
		IF dly.Q OR Refresh_Now THEN
			dly.PT:=Refresh_Period;
			Refresh_Now:=FALSE;
			sta:=1;
		END_IF

	1: (* === Start update when MB is free *)
		IF NOT (MODBUS.MB_Lock OR MODBUS.MB_Start) THEN
			MODBUS.MB_Lock:=TRUE;
			MODBUS.MB_Query.SlaveAddress:=ADDRESS;
			MODBUS.MB_Query.FunctionCode:=16#03;
			(* Start query *)
			MODBUS.MB_Query.Read_StartAddress:=16#1000;
			MODBUS.MB_Query.Read_Quantity:=16#16;
			MODBUS.MB_Start:=TRUE;
			sta:=2;
		END_IF

	2:	IF NOT MODBUS.MB_Start THEN
			IF MODBUS.MB_MASTER.MB_Error<>MB_NO_ERROR OR MODBUS.MB_Resp.Error<>0 THEN
				sta:=100;
			ELSE
				(* Read response data *)
				COPY_32SWAP16(ADR(MODBUS.MB_Resp.Data[ 0]),ADR(Data.V_3P));
				COPY_32SWAP16(ADR(MODBUS.MB_Resp.Data[ 2]),ADR(Data.V_L1N));
				COPY_32SWAP16(ADR(MODBUS.MB_Resp.Data[ 4]),ADR(Data.V_L2N));
				COPY_32SWAP16(ADR(MODBUS.MB_Resp.Data[ 6]),ADR(Data.V_L3N));
				COPY_32SWAP16(ADR(MODBUS.MB_Resp.Data[ 8]),ADR(Data.V_L1L2));
				COPY_32SWAP16(ADR(MODBUS.MB_Resp.Data[10]),ADR(Data.V_L2L3));
				COPY_32SWAP16(ADR(MODBUS.MB_Resp.Data[12]),ADR(Data.V_L3L1));
				COPY_32SWAP16(ADR(MODBUS.MB_Resp.Data[14]),ADR(Data.I_3P));
				COPY_32SWAP16(ADR(MODBUS.MB_Resp.Data[16]),ADR(Data.I_L1));
				COPY_32SWAP16(ADR(MODBUS.MB_Resp.Data[18]),ADR(Data.I_L2));
				COPY_32SWAP16(ADR(MODBUS.MB_Resp.Data[20]),ADR(Data.I_L3));
				(* Start query *)
				MODBUS.MB_Query.Read_StartAddress:=16#1016;
				MODBUS.MB_Query.Read_Quantity:=16#10;
				MODBUS.MB_Start:=TRUE;
				sta:=3;
			END_IF
		END_IF

	3:	IF NOT MODBUS.MB_Start THEN
			IF MODBUS.MB_MASTER.MB_Error<>MB_NO_ERROR OR MODBUS.MB_Resp.Error<>0 THEN
				sta:=100;
			ELSE
				(* Read response data *)
				COPY_32SWAP16(ADR(MODBUS.MB_Resp.Data[ 0]),ADR(Data.PF_3P));
				COPY_32SWAP16(ADR(MODBUS.MB_Resp.Data[ 2]),ADR(Data.PF_L1));
				COPY_32SWAP16(ADR(MODBUS.MB_Resp.Data[ 4]),ADR(Data.PF_L2));
				COPY_32SWAP16(ADR(MODBUS.MB_Resp.Data[ 6]),ADR(Data.PF_L3));
				COPY_32SWAP16(ADR(MODBUS.MB_Resp.Data[ 8]),ADR(Data.COS_3P));
				COPY_32SWAP16(ADR(MODBUS.MB_Resp.Data[10]),ADR(Data.COS_L1));
				COPY_32SWAP16(ADR(MODBUS.MB_Resp.Data[12]),ADR(Data.COS_L2));
				COPY_32SWAP16(ADR(MODBUS.MB_Resp.Data[14]),ADR(Data.COS_L3));
				(* Start query *)
				MODBUS.MB_Query.Read_StartAddress:=16#1026;
				MODBUS.MB_Query.Read_Quantity:=16#10;
				MODBUS.MB_Start:=TRUE;
				sta:=4;
			END_IF
		END_IF

	4:	IF NOT MODBUS.MB_Start THEN
			IF MODBUS.MB_MASTER.MB_Error<>MB_NO_ERROR OR MODBUS.MB_Resp.Error<>0 THEN
				sta:=100;
			ELSE
				(* Read response data *)
				COPY_32SWAP16(ADR(MODBUS.MB_Resp.Data[ 0]),ADR(Data.PF_3P));
				COPY_32SWAP16(ADR(MODBUS.MB_Resp.Data[ 2]),ADR(Data.PF_L1));
				COPY_32SWAP16(ADR(MODBUS.MB_Resp.Data[ 4]),ADR(Data.PF_L2));
				COPY_32SWAP16(ADR(MODBUS.MB_Resp.Data[ 6]),ADR(Data.PF_L3));
				COPY_32SWAP16(ADR(MODBUS.MB_Resp.Data[ 8]),ADR(Data.COS_3P));
				COPY_32SWAP16(ADR(MODBUS.MB_Resp.Data[10]),ADR(Data.COS_L1));
				COPY_32SWAP16(ADR(MODBUS.MB_Resp.Data[12]),ADR(Data.COS_L2));
				COPY_32SWAP16(ADR(MODBUS.MB_Resp.Data[14]),ADR(Data.COS_L3));
				(* Start query *)
				MODBUS.MB_Query.Read_StartAddress:=16#1026;
				MODBUS.MB_Query.Read_Quantity:=16#10;
				MODBUS.MB_Start:=TRUE;
				sta:=5;
			END_IF
		END_IF

	5:	IF NOT MODBUS.MB_Start THEN
			IF MODBUS.MB_MASTER.MB_Error<>MB_NO_ERROR OR MODBUS.MB_Resp.Error<>0 THEN
				sta:=100;
			ELSE
				(* Read response data *)
				COPY_32SWAP16(ADR(MODBUS.MB_Resp.Data[ 0]),ADR(Data.VA_3P));
				COPY_32SWAP16(ADR(MODBUS.MB_Resp.Data[ 2]),ADR(Data.VA_L1));
				COPY_32SWAP16(ADR(MODBUS.MB_Resp.Data[ 4]),ADR(Data.VA_L2));
				COPY_32SWAP16(ADR(MODBUS.MB_Resp.Data[ 6]),ADR(Data.VA_L3));
				COPY_32SWAP16(ADR(MODBUS.MB_Resp.Data[ 8]),ADR(Data.P_3P));
				COPY_32SWAP16(ADR(MODBUS.MB_Resp.Data[10]),ADR(Data.P_L1));
				COPY_32SWAP16(ADR(MODBUS.MB_Resp.Data[12]),ADR(Data.P_L2));
				COPY_32SWAP16(ADR(MODBUS.MB_Resp.Data[14]),ADR(Data.P_L3));
				(* Start query *)
				MODBUS.MB_Query.Read_StartAddress:=16#1036;
				MODBUS.MB_Query.Read_Quantity:=16#0C;
				MODBUS.MB_Start:=TRUE;
				sta:=6;
			END_IF
		END_IF

	6:	IF NOT MODBUS.MB_Start THEN
			IF MODBUS.MB_MASTER.MB_Error<>MB_NO_ERROR OR MODBUS.MB_Resp.Error<>0 THEN
				sta:=100;
			ELSE
				(* Read response data *)
				COPY_32SWAP16(ADR(MODBUS.MB_Resp.Data[ 0]),ADR(Data.Q_3P));
				COPY_32SWAP16(ADR(MODBUS.MB_Resp.Data[ 2]),ADR(Data.Q_L1));
				COPY_32SWAP16(ADR(MODBUS.MB_Resp.Data[ 4]),ADR(Data.Q_L2));
				COPY_32SWAP16(ADR(MODBUS.MB_Resp.Data[ 6]),ADR(Data.Q_L3));
				COPY_32SWAP16(ADR(MODBUS.MB_Resp.Data[ 8]),ADR(Data.WH_3P));
				COPY_32SWAP16(ADR(MODBUS.MB_Resp.Data[10]),ADR(Data.VARH_3P));
				(* Start query *)
				MODBUS.MB_Query.Read_StartAddress:=16#1046;
				MODBUS.MB_Query.Read_Quantity:=16#02;
				MODBUS.MB_Start:=TRUE;
				sta:=7;
			END_IF
		END_IF

	7:	IF NOT MODBUS.MB_Start THEN
			IF MODBUS.MB_MASTER.MB_Error<>MB_NO_ERROR OR MODBUS.MB_Resp.Error<>0 THEN
				sta:=100;
			ELSE
				(* Read response data *)
				COPY_32SWAP16(ADR(MODBUS.MB_Resp.Data[ 0]),ADR(Data.FREQ));
				(* Start query *)
				MODBUS.MB_Query.Read_StartAddress:=16#1060;
				MODBUS.MB_Query.Read_Quantity:=16#0A;
				MODBUS.MB_Start:=TRUE;
				sta:=8;
			END_IF
		END_IF

	8:	IF NOT MODBUS.MB_Start THEN
			IF MODBUS.MB_MASTER.MB_Error<>MB_NO_ERROR OR MODBUS.MB_Resp.Error<>0 THEN
				sta:=100;
			ELSE
				(* Read response data *)
				COPY_32SWAP16(ADR(MODBUS.MB_Resp.Data[ 0]),ADR(Data.I_L1_Max));
				COPY_32SWAP16(ADR(MODBUS.MB_Resp.Data[ 2]),ADR(Data.I_L2_Max));
				COPY_32SWAP16(ADR(MODBUS.MB_Resp.Data[ 4]),ADR(Data.I_L3_Max));
				COPY_32SWAP16(ADR(MODBUS.MB_Resp.Data[ 6]),ADR(Data.P_3P_Max));
				COPY_32SWAP16(ADR(MODBUS.MB_Resp.Data[ 8]),ADR(Data.Q_3P_Max));
				(* Start query *)
				MODBUS.MB_Query.Read_StartAddress:=16#1070;
				MODBUS.MB_Query.Read_Quantity:=16#02;
				MODBUS.MB_Start:=TRUE;
				sta:=9;
			END_IF
		END_IF

	9:	IF NOT MODBUS.MB_Start THEN
			IF MODBUS.MB_MASTER.MB_Error<>MB_NO_ERROR OR MODBUS.MB_Resp.Error<>0 THEN
				sta:=100;
			ELSE
				(* Read response data *)
				COPY_32SWAP16(ADR(MODBUS.MB_Resp.Data[ 0]),ADR(Data.P_3P_Avg15m));
				(* Release MODBUS *)
				MODBUS.MB_Lock:=FALSE;
				(* Update status *)
				Status_Log:=0;
				Status_Vis:=16#20F020;
				sta:=0;
			END_IF
		END_IF

	100: (* === Check MODBUS error *)
		MODBUS.MB_Lock:=FALSE;
		Status_Log:=2;
		Status_Vis:=16#2020F0;
		sta:=0;

ELSE
	sta:=0;
END_CASE
END_FUNCTION_BLOCK

(* POU Plant_Objects/obj_MODBUS_ELGAS_MINIELCOR, ST *)
FUNCTION_BLOCK obj_MODBUS_ELGAS_MINIELCOR
VAR_INPUT
	(* Settings *)
	ID				: BYTE;
	ADDRESS			: BYTE:=1;
(*	Refresh_Period	: TIME:=t#1m30s;*)
	Refresh_Time	: BYTE:=90;
	(* Controls *)
(*	Refresh_Auto	: BOOL; (* Enable automatic refresh *)*)
(*	Refresh_Now		: BOOL; (* Force an immediate refresh *)*)
END_VAR
VAR_IN_OUT
	MODBUS			: obj_MODBUS;
END_VAR
VAR_OUTPUT
	Data			: typ_MODBUS_ELGAS_MINIELCOR;
	(* Status *)
	Status_Log		: BYTE;
	Status_Vis 		: DWORD;
END_VAR
VAR
	dly 	 : TON := (PT:=t#5s);
	sta		 : BYTE; (* Status *)

	addr : WORD:=19;
	siz: WORD:=2;

END_VAR
CASE sta OF

	0: (* === Initialize *)

		MODBUS.VARS[0].SlaveAddress:=1;
		MODBUS.VARS[0].FunCode:=3;
		MODBUS.VARS[0].FunAddress:=3;
		MODBUS.VARS[0].Refresh_Time:=Refresh_Time;
		MODBUS.VARS[0].Variable_Mirror:=0;
		MODBUS.VARS[0].Variable_Size:=4;
		MODBUS.VARS[0].Variable:=ADR(Data.Vb);

		MODBUS.VARS[1].SlaveAddress:=1;
		MODBUS.VARS[1].FunCode:=3;
		MODBUS.VARS[1].FunAddress:=19;
		MODBUS.VARS[1].Refresh_Time:=Refresh_Time;
		MODBUS.VARS[1].Variable_Mirror:=0;
		MODBUS.VARS[1].Variable_Size:=200;
		MODBUS.VARS[1].Variable:=ADR(Data.Vm);

		MODBUS.VARS[2].SlaveAddress:=1;
		MODBUS.VARS[2].FunCode:=3;
		MODBUS.VARS[2].FunAddress:=25;
		MODBUS.VARS[2].Refresh_Time:=Refresh_Time;
		MODBUS.VARS[2].Variable_Mirror:=0;
		MODBUS.VARS[2].Variable_Size:=200;
		MODBUS.VARS[2].Variable:=ADR(Data.P);

		MODBUS.VARS[3].SlaveAddress:=1;
		MODBUS.VARS[3].FunCode:=3;
		MODBUS.VARS[3].FunAddress:=27;
		MODBUS.VARS[3].Refresh_Time:=Refresh_Time;
		MODBUS.VARS[3].Variable_Mirror:=0;
		MODBUS.VARS[3].Variable_Size:=200;
		MODBUS.VARS[3].Variable:=ADR(Data.T);

		MODBUS.VARS[4].SlaveAddress:=1;
		MODBUS.VARS[4].FunCode:=3;
		MODBUS.VARS[4].FunAddress:=39;
		MODBUS.VARS[4].Refresh_Time:=Refresh_Time;
		MODBUS.VARS[4].Variable_Mirror:=0;
		MODBUS.VARS[4].Variable_Size:=200;
		MODBUS.VARS[4].Variable:=ADR(Data.C);

		MODBUS.VARS[5].SlaveAddress:=1;
		MODBUS.VARS[5].FunCode:=3;
		MODBUS.VARS[5].FunAddress:=7;
		MODBUS.VARS[5].Refresh_Time:=Refresh_Time;
		MODBUS.VARS[5].Variable_Mirror:=0;
		MODBUS.VARS[5].Variable_Size:=4;
		MODBUS.VARS[5].Variable:=ADR(Data.Vbs);

		MODBUS.VARS[6].SlaveAddress:=1;
		MODBUS.VARS[6].FunCode:=3;
		MODBUS.VARS[6].FunAddress:=11;
		MODBUS.VARS[6].Refresh_Time:=Refresh_Time;
		MODBUS.VARS[6].Variable_Mirror:=0;
		MODBUS.VARS[6].Variable_Size:=4;
		MODBUS.VARS[6].Variable:=ADR(Data.Vb_d_d);

		MODBUS.VARS[7].SlaveAddress:=1;
		MODBUS.VARS[7].FunCode:=3;
		MODBUS.VARS[7].FunAddress:=15;
		MODBUS.VARS[7].Refresh_Time:=Refresh_Time;
		MODBUS.VARS[7].Variable_Mirror:=0;
		MODBUS.VARS[7].Variable_Size:=4;
		MODBUS.VARS[7].Variable:=ADR(Data.Vb_d_m);

		MODBUS.VARS[8].SlaveAddress:=1;
		MODBUS.VARS[8].FunCode:=3;
		MODBUS.VARS[8].FunAddress:=21;
		MODBUS.VARS[8].Refresh_Time:=Refresh_Time;
		MODBUS.VARS[8].Variable_Mirror:=0;
		MODBUS.VARS[8].Variable_Size:=200;
		MODBUS.VARS[8].Variable:=ADR(Data.Vm_d_d);

		MODBUS.VARS[9].SlaveAddress:=1;
		MODBUS.VARS[9].FunCode:=3;
		MODBUS.VARS[9].FunAddress:=31;
		MODBUS.VARS[9].Refresh_Time:=Refresh_Time;
		MODBUS.VARS[9].Variable_Mirror:=0;
		MODBUS.VARS[9].Variable_Size:=200;
		MODBUS.VARS[9].Variable:=ADR(Data.BC_EVC);

		MODBUS.VARS[10].SlaveAddress:=1;
		MODBUS.VARS[10].FunCode:=3;
		MODBUS.VARS[10].FunAddress:=29;
		MODBUS.VARS[10].Refresh_Time:=Refresh_Time;
		MODBUS.VARS[10].Variable_Mirror:=0;
		MODBUS.VARS[10].Variable_Size:=200;
		MODBUS.VARS[10].Variable:=ADR(Data.BV_EVC);

		MODBUS.VARS[11].SlaveAddress:=1;
		MODBUS.VARS[11].FunCode:=3;
		MODBUS.VARS[11].FunAddress:=35;
		MODBUS.VARS[11].Refresh_Time:=Refresh_Time;
		MODBUS.VARS[11].Variable_Mirror:=0;
		MODBUS.VARS[11].Variable_Size:=200;
		MODBUS.VARS[11].Variable:=ADR(Data.Q);

		MODBUS.VARS[12].SlaveAddress:=1;
		MODBUS.VARS[12].FunCode:=3;
		MODBUS.VARS[12].FunAddress:=37;
		MODBUS.VARS[12].Refresh_Time:=Refresh_Time;
		MODBUS.VARS[12].Variable_Mirror:=0;
		MODBUS.VARS[12].Variable_Size:=200;
		MODBUS.VARS[12].Variable:=ADR(Data.Qb);

		MODBUS.VARS[13].SlaveAddress:=1;
		MODBUS.VARS[13].FunCode:=3;
		MODBUS.VARS[13].FunAddress:=55;
		MODBUS.VARS[13].Refresh_Time:=Refresh_Time;
		MODBUS.VARS[13].Variable_Mirror:=0;
		MODBUS.VARS[13].Variable_Size:=1;
		MODBUS.VARS[13].Variable:=ADR(Data.D_Err);

		MODBUS.VARS[14].SlaveAddress:=1;
		MODBUS.VARS[14].FunCode:=3;
		MODBUS.VARS[14].FunAddress:=56;
		MODBUS.VARS[14].Refresh_Time:=Refresh_Time;
		MODBUS.VARS[14].Variable_Mirror:=0;
		MODBUS.VARS[14].Variable_Size:=200;
		MODBUS.VARS[14].Variable:=ADR(Data.Status);

		MODBUS.VARS_En:=TRUE;

		sta:=1;

	1:	(* === Check status *)
		IF MODBUS.VARS_Alarm OR Data.D_Err<>0 THEN
			Status_Log:=2;
			Status_Vis:=16#2020F0;
		ELSE
			Status_Log:=0;
			Status_Vis:=16#20F020;
		END_IF


(*
	1: (* === Wait update signals *)
		dly(IN:=NOT (dly.Q OR Refresh_Now OR (NOT Refresh_Auto)));
		IF dly.Q OR Refresh_Now THEN
			dly.PT:=Refresh_Period;
			Refresh_Now:=FALSE;
			sta:=2;
		END_IF

	2: (* === Start update when MB is free *)
		IF NOT (MODBUS.MB_Lock OR MODBUS.MB_Start) THEN
			MODBUS.MB_Lock:=TRUE;
			MODBUS.MB_Query.SlaveAddress:=ADDRESS;
			MODBUS.MB_Query.FunctionCode:=16#03;
			(* Start query *)
			MODBUS.MB_Query.Read_StartAddress:=addr;
			MODBUS.MB_Query.Read_Quantity:=siz;
			MODBUS.MB_Start:=TRUE;
			sta:=10;
		END_IF

